KUKA KRL program: MyProgram_345().src

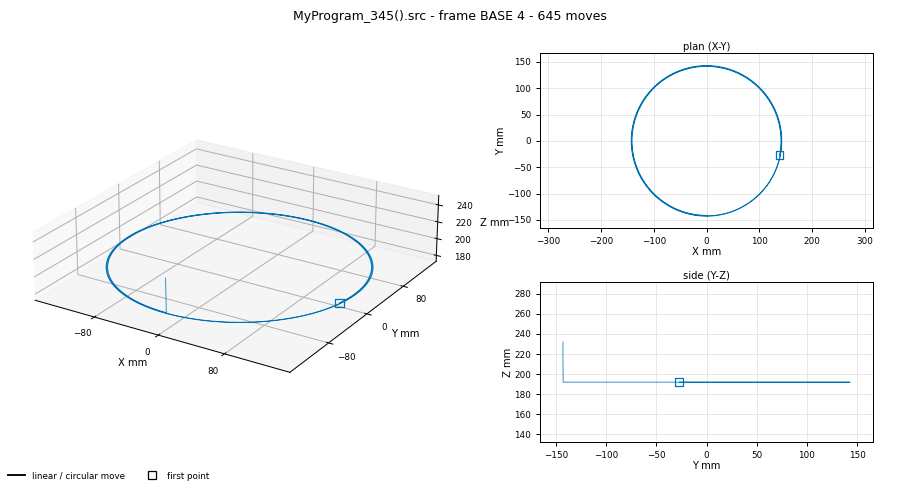
[picture p0: tool path of MyProgram_345().src in frame BASE 4, 645 of 645 moves have a stored position in this frame; points joined in program order, loops and branches not executed]
&ACCESS RVP
&REL 1
&PARAM TEMPLATE = C:\KRC\Roboter\Template\vorgabe
&PARAM EDITMASK = *
DEF MyProgram_345()
; ---- Setting reference (Base) ----
$BASE = BASE_DATA[4]

; --------------------------
; ---- Setting tool (TCP) ----
$TOOL = TOOL_DATA[3]
; --------------------------

$VEL.CP = VEL_APROX_PRINT
Startdeposition()
$VEL.CP = VEL_PRINT
LIN {X 138.5242,Y -27.3155,Z 192,A -4.5252,B 0.5611,C 0.0605,E1 0.722,E2 458.3283} C_DIS
LIN {X 139.2365,Y -23.4021,Z 192,A -3.481,B 0.5613,C 0.0586,E1 0.7225,E2 457.3622} C_DIS
LIN {X 139.7745,Y -19.9386,Z 192,A -2.1592,B 0.5617,C 0.0551,E1 0.7231,E2 456.0535} C_DIS
LIN {X 140.2586,Y -16.1943,Z 192,A -0.8679,B 0.562,C 0.052,E1 0.7235,E2 454.7945} C_DIS
LIN {X 140.6407,Y -12.4489,Z 192,A 0.376,B 0.5622,C 0.049,E1 0.7238,E2 453.5886} C_DIS
LIN {X 140.9254,Y -8.6325,Z 192,A 1.5623,B 0.5625,C 0.0463,E1 0.724,E2 452.4515} C_DIS
LIN {X 141.1118,Y -4.7394,Z 192,A 2.9278,B 0.5627,C 0.0429,E1 0.7241,E2 451.1146} C_DIS
LIN {X 141.1896,Y -0.6145,Z 192,A 4.1944,B 0.563,C 0.04,E1 0.7241,E2 449.9021} C_DIS
LIN {X 141.1462,Y 3.5236,Z 192,A 5.5812,B 0.5632,C 0.0366,E1 0.7241,E2 448.5537} C_DIS
LIN {X 140.9906,Y 7.504,Z 192,A 6.8322,B 0.5634,C 0.0338,E1 0.724,E2 447.3507} C_DIS
LIN {X 140.737,Y 11.3097,Z 192,A 8.1166,B 0.5635,C 0.0306,E1 0.7237,E2 446.1005} C_DIS
LIN {X 140.4091,Y 14.8267,Z 192,A 9.1787,B 0.5637,C 0.0283,E1 0.7234,E2 445.0867} C_DIS
LIN {X 140.0043,Y 18.2549,Z 192,A 10.3048,B 0.5637,C 0.0256,E1 0.7231,E2 443.996} C_DIS
LIN {X 139.3324,Y 22.8275,Z 192,A 12.3132,B 0.564,C 0.0198,E1 0.7222,E2 441.9693} C_DIS
LIN {X 138.4504,Y 27.6793,Z 192,A 14.134,B 0.5642,C 0.0151,E1 0.7212,E2 440.1713} C_DIS
LIN {X 137.041,Y 33.9819,Z 192,A 15.5668,B 0.5642,C 0.0131,E1 0.7204,E2 438.8911} C_DIS
LIN {X 135.2457,Y 40.5419,Z 192,A 17.9276,B 0.5643,C 0.0072,E1 0.7186,E2 436.5801} C_DIS
LIN {X 134.1293,Y 44.0907,Z 192,A 19.1032,B 0.5643,C 0.0045,E1 0.7176,E2 435.4462} C_DIS
LIN {X 132.9221,Y 47.6043,Z 192,A 20.2677,B 0.5643,C 0.0019,E1 0.7166,E2 434.3242} C_DIS
LIN {X 131.6486,Y 51.0197,Z 192,A 21.3577,B 0.5643,C -0.0004,E1 0.7155,E2 433.2822} C_DIS
LIN {X 130.3439,Y 54.2664,Z 192,A 22.5748,B 0.5643,C -0.0033,E1 0.7143,E2 432.0898} C_DIS
LIN {X 129.2468,Y 56.8363,Z 192,A 23.7777,B 0.5643,C -0.0067,E1 0.7129,E2 430.8782} C_DIS
LIN {X 127.791,Y 60.0377,Z 192,A 24.7987,B 0.5643,C -0.0087,E1 0.7118,E2 429.9068} C_DIS
LIN {X 126.0848,Y 63.5397,Z 192,A 26.0063,B 0.5643,C -0.0113,E1 0.7103,E2 428.7443} C_DIS
LIN {X 124.1773,Y 67.1944,Z 192,A 27.4129,B 0.5642,C -0.0146,E1 0.7085,E2 427.3696} C_DIS
LIN {X 122.0387,Y 71.0039,Z 192,A 28.7948,B 0.5641,C -0.0176,E1 0.7066,E2 426.0344} C_DIS
LIN {X 119.7699,Y 74.767,Z 192,A 30.2924,B 0.564,C -0.021,E1 0.7045,E2 424.5706} C_DIS
LIN {X 117.2837,Y 78.6098,Z 192,A 31.8113,B 0.5638,C -0.0243,E1 0.7022,E2 423.0915} C_DIS
LIN {X 114.6921,Y 82.3449,Z 192,A 33.3322,B 0.5637,C -0.0277,E1 0.6998,E2 421.6084} C_DIS
LIN {X 111.9551,Y 86.0294,Z 192,A 35.0251,B 0.5635,C -0.0316,E1 0.6969,E2 419.9352} C_DIS
LIN {X 109.8588,Y 88.6901,Z 192,A 35.9356,B 0.5634,C -0.0331,E1 0.6954,E2 419.0784} C_DIS
LIN {X 107.1281,Y 91.9702,Z 192,A 37.4224,B 0.5632,C -0.0364,E1 0.6927,E2 417.6197} C_DIS
LIN {X 104.0065,Y 95.4859,Z 192,A 38.9764,B 0.563,C -0.0395,E1 0.6899,E2 416.106} C_DIS
LIN {X 101.0756,Y 98.5838,Z 192,A 40.4488,B 0.5628,C -0.0426,E1 0.687,E2 414.6629} C_DIS
LIN {X 98.9534,Y 100.7132,Z 192,A 41.7136,B 0.5625,C -0.0455,E1 0.6845,E2 413.3929} C_DIS
LIN {X 95.9465,Y 103.5824,Z 192,A 42.79,B 0.5625,C -0.0471,E1 0.6824,E2 412.3852} C_DIS
LIN {X 93.0608,Y 106.1823,Z 192,A 44.1725,B 0.5622,C -0.05,E1 0.6795,E2 411.0242} C_DIS
LIN {X 89.4357,Y 109.2528,Z 192,A 45.7484,B 0.5619,C -0.0529,E1 0.6761,E2 409.4873} C_DIS
LIN {X 86.0148,Y 111.9663,Z 192,A 47.2728,B 0.5616,C -0.0558,E1 0.6728,E2 407.9901} C_DIS
LIN {X 82.3075,Y 114.7189,Z 192,A 48.8316,B 0.5613,C -0.0587,E1 0.6693,E2 406.4657} C_DIS
LIN {X 78.8287,Y 117.137,Z 192,A 50.2736,B 0.561,C -0.0612,E1 0.666,E2 405.0538} C_DIS
LIN {X 75.018,Y 119.6134,Z 192,A 51.8114,B 0.5607,C -0.0639,E1 0.6623,E2 403.549} C_DIS
LIN {X 71.2617,Y 121.8883,Z 192,A 53.3553,B 0.5604,C -0.0666,E1 0.6586,E2 402.0307} C_DIS
LIN {X 67.3753,Y 124.0788,Z 192,A 54.905,B 0.5601,C -0.0691,E1 0.6548,E2 400.5088} C_DIS
LIN {X 62.4464,Y 126.6285,Z 192,A 56.6735,B 0.5598,C -0.0718,E1 0.6504,E2 398.7912} C_DIS
LIN {X 59.695,Y 127.9495,Z 192,A 57.8562,B 0.5595,C -0.0738,E1 0.6474,E2 397.6145} C_DIS
LIN {X 56.3645,Y 129.4508,Z 192,A 59.1231,B 0.5593,C -0.0757,E1 0.6441,E2 396.3702} C_DIS
LIN {X 53.5399,Y 130.6464,Z 192,A 60.313,B 0.559,C -0.0776,E1 0.641,E2 395.1862} C_DIS
LIN {X 49.9685,Y 132.052,Z 192,A 61.5782,B 0.5588,C -0.0793,E1 0.6377,E2 393.9512} C_DIS
LIN {X 46.7273,Y 133.2336,Z 192,A 62.8545,B 0.5585,C -0.0811,E1 0.6342,E2 392.6878} C_DIS
LIN {X 43.1768,Y 134.4254,Z 192,A 64.2206,B 0.5582,C -0.083,E1 0.6306,E2 391.3377} C_DIS
LIN {X 35.1127,Y 136.754,Z 192,A 67.1312,B 0.5577,C -0.0866,E1 0.6226,E2 388.478} C_DIS
LIN {X 28.547,Y 138.2738,Z 192,A 69.6083,B 0.5572,C -0.0895,E1 0.6157,E2 386.0273} C_DIS
LIN {X 23.8823,Y 139.1564,Z 192,A 71.397,B 0.5569,C -0.0915,E1 0.6107,E2 384.2529} C_DIS
LIN {X 20.3949,Y 139.7092,Z 192,A 72.6632,B 0.5567,C -0.0928,E1 0.6071,E2 383.0035} C_DIS
LIN {X 17.2318,Y 140.1349,Z 192,A 73.8305,B 0.5565,C -0.0939,E1 0.6038,E2 381.8492} C_DIS
LIN {X 13.6174,Y 140.5313,Z 192,A 75.1425,B 0.5563,C -0.0951,E1 0.6001,E2 380.5536} C_DIS
LIN {X 9.6219,Y 140.8628,Z 192,A 76.7148,B 0.5561,C -0.0966,E1 0.5955,E2 378.9872} C_DIS
LIN {X 5.5113,Y 141.0819,Z 192,A 78.1803,B 0.5559,C -0.0977,E1 0.5913,E2 377.5421} C_DIS
LIN {X 1.1101,Y 141.1856,Z 192,A 79.8215,B 0.5556,C -0.0988,E1 0.5866,E2 375.9156} C_DIS
LIN {X -2.5499,Y 141.1667,Z 192,A 81.2212,B 0.5555,C -0.0998,E1 0.5826,E2 374.5247} C_DIS
LIN {X -6.4253,Y 141.0448,Z 192,A 82.7609,B 0.5553,C -0.1008,E1 0.5781,E2 372.9889} C_DIS
LIN {X -10.1902,Y 140.8213,Z 192,A 84.1527,B 0.5552,C -0.1015,E1 0.5741,E2 371.6108} C_DIS
LIN {X -13.9892,Y 140.4956,Z 192,A 85.4332,B 0.5551,C -0.102,E1 0.5705,E2 370.3563} C_DIS
LIN {X -18.5339,Y 139.9678,Z 192,A 87.497,B 0.5549,C -0.1031,E1 0.5645,E2 368.2736} C_DIS
LIN {X -22.8627,Y 139.3265,Z 192,A 89.1306,B 0.5548,C -0.1036,E1 0.5598,E2 366.6543} C_DIS
LIN {X -26.405,Y 138.6983,Z 192,A 90.5233,B 0.5548,C -0.1039,E1 0.5559,E2 365.2685} C_DIS
LIN {X -29.884,Y 137.9904,Z 192,A 91.948,B 0.5547,C -0.1042,E1 0.5518,E2 363.846} C_DIS
LIN {X -33.9548,Y 137.0478,Z 192,A 93.7775,B 0.5546,C -0.1046,E1 0.5466,E2 362.0046} C_DIS
LIN {X -38.0062,Y 135.9776,Z 192,A 95.319,B 0.5546,C -0.1046,E1 0.5423,E2 360.4788} C_DIS
LIN {X -41.3069,Y 135.0115,Z 192,A 96.5979,B 0.5546,C -0.1044,E1 0.5388,E2 359.2116} C_DIS
LIN {X -44.3383,Y 134.0469,Z 192,A 97.9917,B 0.5546,C -0.1044,E1 0.5349,E2 357.8086} C_DIS
LIN {X -47.0982,Y 133.1045,Z 192,A 99.3629,B 0.5546,C -0.1044,E1 0.5311,E2 356.4203} C_DIS
LIN {X -50.6134,Y 131.8066,Z 192,A 100.8481,B 0.5547,C -0.104,E1 0.527,E2 354.9391} C_DIS
LIN {X -53.6288,Y 130.6102,Z 192,A 102.5352,B 0.5547,C -0.1038,E1 0.5224,E2 353.2173} C_DIS
LIN {X -57.197,Y 129.0856,Z 192,A 103.7496,B 0.5549,C -0.1031,E1 0.5193,E2 352.038} C_DIS
LIN {X -60.1404,Y 127.7424,Z 192,A 105.2375,B 0.5549,C -0.1026,E1 0.5153,E2 350.5342} C_DIS
LIN {X -64.6568,Y 125.516,Z 192,A 107.3683,B 0.5552,C -0.1015,E1 0.5097,E2 348.396} C_DIS
LIN {X -67.4098,Y 124.06,Z 192,A 109.262,B 0.5552,C -0.1009,E1 0.5048,E2 346.4422} C_DIS
LIN {X -71.8848,Y 121.5223,Z 192,A 110.9515,B 0.5556,C -0.0993,E1 0.5006,E2 344.7923} C_DIS
LIN {X -75.7994,Y 119.1197,Z 192,A 112.9667,B 0.5558,C -0.0978,E1 0.4956,E2 342.7635} C_DIS
LIN {X -79.6799,Y 116.5594,Z 192,A 115.3227,B 0.5561,C -0.0961,E1 0.4899,E2 340.3627} C_DIS
LIN {X -82.7739,Y 114.3826,Z 192,A 116.7096,B 0.5564,C -0.0946,E1 0.4866,E2 338.9912} C_DIS
LIN {X -86.4509,Y 111.6295,Z 192,A 118.7765,B 0.5567,C -0.0925,E1 0.4818,E2 336.9053} C_DIS
LIN {X -90.153,Y 108.6616,Z 192,A 120.8713,B 0.5571,C -0.0902,E1 0.4771,E2 334.7948} C_DIS
LIN {X -93.2484,Y 106.0177,Z 192,A 122.8335,B 0.5575,C -0.088,E1 0.4728,E2 332.8028} C_DIS
LIN {X -96.6151,Y 102.959,Z 192,A 124.9266,B 0.5579,C -0.0854,E1 0.4683,E2 330.686} C_DIS
LIN {X -99.7496,Y 99.9251,Z 192,A 126.9433,B 0.5583,C -0.0827,E1 0.4641,E2 328.6454} C_DIS
LIN {X -102.8714,Y 96.708,Z 192,A 129.0955,B 0.5587,C -0.0797,E1 0.4598,E2 326.4604} C_DIS
LIN {X -105.9836,Y 93.287,Z 192,A 131.2873,B 0.5592,C -0.0764,E1 0.4555,E2 324.2373} C_DIS
LIN {X -108.8114,Y 89.9722,Z 192,A 133.4193,B 0.5596,C -0.073,E1 0.4515,E2 322.0688} C_DIS
LIN {X -111.9551,Y 86.0294,Z 192,A 136.4707,B 0.5602,C -0.0683,E1 0.446,E2 318.9128} C_DIS
LIN {X -114.7818,Y 82.2196,Z 192,A 138.1377,B 0.5606,C -0.065,E1 0.4432,E2 317.2743} C_DIS
LIN {X -117.5668,Y 78.1857,Z 192,A 140.6425,B 0.5611,C -0.0605,E1 0.4391,E2 314.7156} C_DIS
LIN {X -119.9857,Y 74.4203,Z 192,A 142.6975,B 0.5615,C -0.0565,E1 0.4359,E2 312.636} C_DIS
LIN {X -123.2884,Y 68.8117,Z 192,A 146.2773,B 0.5622,C -0.0496,E1 0.4307,E2 308.9552} C_DIS
LIN {X -125.6023,Y 64.4874,Z 192,A 148.651,B 0.5626,C -0.0446,E1 0.4275,E2 306.5401} C_DIS
LIN {X -127.9588,Y 59.6746,Z 192,A 151.6555,B 0.5631,C -0.0383,E1 0.4237,E2 303.4432} C_DIS
LIN {X -129.8067,Y 55.5407,Z 192,A 154.0352,B 0.5634,C -0.0331,E1 0.421,E2 301.0026} C_DIS
LIN {X -131.5415,Y 51.2953,Z 192,A 155.8705,B 0.5636,C -0.0286,E1 0.419,E2 299.1713} C_DIS
LIN {X -132.5169,Y 48.7273,Z 192,A 157.7152,B 0.5638,C -0.0246,E1 0.4171,E2 297.2425} C_DIS
LIN {X -133.9593,Y 44.6014,Z 192,A 159.9336,B 0.564,C -0.0194,E1 0.4151,E2 294.9728} C_DIS
LIN {X -134.9324,Y 41.5656,Z 192,A 161.7041,B 0.5642,C -0.0153,E1 0.4135,E2 293.1463} C_DIS
LIN {X -135.8406,Y 38.4962,Z 192,A 163.2032,B 0.5642,C -0.0115,E1 0.4123,E2 291.6241} C_DIS
LIN {X -136.6138,Y 35.6597,Z 192,A 165.5888,B 0.5643,C -0.0063,E1 0.4106,E2 289.0943} C_DIS
LIN {X -137.591,Y 31.6731,Z 192,A 166.8745,B 0.5643,C -0.0025,E1 0.4097,E2 287.8561} C_DIS
LIN {X -138.5269,Y 27.3017,Z 192,A 169.7946,B 0.5643,C 0.0043,E1 0.408,E2 284.8005} C_DIS
LIN {X -139.6213,Y 20.9931,Z 192,A 173.1218,B 0.5643,C 0.0128,E1 0.4064,E2 281.3831} C_DIS
LIN {X -140.228,Y 16.451,Z 192,A 175.5869,B 0.5641,C 0.019,E1 0.4055,E2 278.8419} C_DIS
LIN {X -140.6546,Y 12.2842,Z 192,A 178.0252,B 0.5638,C 0.0251,E1 0.4049,E2 276.3092} C_DIS
LIN {X -140.8877,Y 9.2448,Z 192,A -179.8372,B 0.5636,C 0.0302,E1 0.4045,E2 274.0544} C_DIS
LIN {X -141.0977,Y 5.1076,Z 192,A -178.0006,B 0.5633,C 0.0352,E1 0.4043,E2 272.1982} C_DIS
LIN {X -141.1833,Y -1.537,Z 192,A -174.4443,B 0.5626,C 0.0443,E1 0.4043,E2 268.5288} C_DIS
LIN {X -141.0589,Y -6.1025,Z 192,A -171.3976,B 0.562,C 0.0516,E1 0.4046,E2 265.321} C_DIS
LIN {X -140.8113,Y -10.3266,Z 192,A -168.6963,B 0.5614,C 0.0581,E1 0.4052,E2 262.4846} C_DIS
LIN {X -140.2534,Y -16.2384,Z 192,A -166.4993,B 0.5607,C 0.0644,E1 0.4058,E2 260.3184} C_DIS
LIN {X -139.8061,Y -19.7168,Z 192,A -164.5222,B 0.5601,C 0.0692,E1 0.4066,E2 258.2647} C_DIS
LIN {X -138.8649,Y -25.5228,Z 192,A -161.2506,B 0.5591,C 0.0772,E1 0.4082,E2 254.8696} C_DIS
LIN {X -138.0677,Y -29.5261,Z 192,A -159.1217,B 0.5583,C 0.0824,E1 0.4095,E2 252.6741} C_DIS
LIN {X -137.2735,Y -33.0212,Z 192,A -157.251,B 0.5576,C 0.0869,E1 0.4107,E2 250.7444} C_DIS
LIN {X -136.3362,Y -36.7007,Z 192,A -155.2273,B 0.5569,C 0.0916,E1 0.4122,E2 248.6517} C_DIS
LIN {X -135.1685,Y -40.794,Z 192,A -152.8988,B 0.556,C 0.097,E1 0.4141,E2 246.2365} C_DIS
LIN {X -134.1293,Y -44.0907,Z 192,A -150.6088,B 0.5551,C 0.1018,E1 0.4162,E2 243.8168} C_DIS
LIN {X -132.8674,Y -47.7561,Z 192,A -149.3984,B 0.5545,C 0.1052,E1 0.4173,E2 242.6605} C_DIS
LIN {X -131.7622,Y -50.7275,Z 192,A -147.3606,B 0.5537,C 0.1093,E1 0.4194,E2 240.5122} C_DIS
LIN {X -130.6124,Y -53.6235,Z 192,A -145.81,B 0.553,C 0.1127,E1 0.4211,E2 238.9196} C_DIS
LIN {X -128.8353,Y -57.7566,Z 192,A -143.4773,B 0.552,C 0.1176,E1 0.4238,E2 236.5116} C_DIS
LIN {X -127.4653,Y -60.7203,Z 192,A -141.7834,B 0.5512,C 0.1211,E1 0.4259,E2 234.7627} C_DIS
LIN {X -125.8921,Y -63.9181,Z 192,A -140.0703,B 0.5504,C 0.1246,E1 0.4282,E2 233.0098} C_DIS
LIN {X -124.1723,Y -67.2036,Z 192,A -137.9104,B 0.5495,C 0.1286,E1 0.4312,E2 230.7509} C_DIS
LIN {X -121.9679,Y -71.1262,Z 192,A -135.6323,B 0.5485,C 0.1329,E1 0.4345,E2 228.4043} C_DIS
LIN {X -119.5569,Y -75.1076,Z 192,A -133.347,B 0.5475,C 0.1371,E1 0.438,E2 226.0584} C_DIS
LIN {X -117.1181,Y -78.8567,Z 192,A -131.1217,B 0.5465,C 0.1409,E1 0.4416,E2 223.7703} C_DIS
LIN {X -114.5576,Y -82.5325,Z 192,A -129.0173,B 0.5456,C 0.1445,E1 0.4451,E2 221.6218} C_DIS
LIN {X -109.5938,Y -89.0184,Z 192,A -124.9502,B 0.5439,C 0.1508,E1 0.4525,E2 217.4383} C_DIS
LIN {X -105.9183,Y -93.3609,Z 192,A -122.2264,B 0.5428,C 0.1547,E1 0.4577,E2 214.6496} C_DIS
LIN {X -102.9112,Y -96.6658,Z 192,A -120.1081,B 0.5419,C 0.1575,E1 0.4619,E2 212.4835} C_DIS
LIN {X -96.5479,Y -103.0223,Z 192,A -115.9063,B 0.5404,C 0.1627,E1 0.4707,E2 208.1948} C_DIS
LIN {X -93.1478,Y -106.1064,Z 192,A -113.9445,B 0.5397,C 0.165,E1 0.475,E2 206.2172} C_DIS
LIN {X -89.5276,Y -109.1777,Z 192,A -111.6621,B 0.539,C 0.1672,E1 0.4802,E2 203.8783} C_DIS
LIN {X -86.0232,Y -111.9598,Z 192,A -109.6421,B 0.5384,C 0.1691,E1 0.4849,E2 201.8256} C_DIS
LIN {X -82.3935,Y -114.6574,Z 192,A -107.5945,B 0.5379,C 0.1709,E1 0.4897,E2 199.7438} C_DIS
LIN {X -78.7099,Y -117.2169,Z 192,A -105.619,B 0.5374,C 0.1724,E1 0.4945,E2 197.7432} C_DIS
LIN {X -75.0257,Y -119.6086,Z 192,A -103.6912,B 0.537,C 0.1737,E1 0.4993,E2 195.7919} C_DIS
LIN {X -71.1828,Y -121.9346,Z 192,A -101.7704,B 0.5366,C 0.1749,E1 0.5041,E2 193.8549} C_DIS
LIN {X -67.3853,Y -124.0734,Z 192,A -99.7334,B 0.5363,C 0.1758,E1 0.5094,E2 191.7744} C_DIS
LIN {X -62.7554,Y -126.4761,Z 192,A -97.6185,B 0.5359,C 0.1769,E1 0.5149,E2 189.6592} C_DIS
LIN {X -58.5907,Y -128.4601,Z 192,A -95.6908,B 0.5357,C 0.1776,E1 0.52,E2 187.7221} C_DIS
LIN {X -54.4999,Y -130.2463,Z 192,A -93.9571,B 0.5355,C 0.1783,E1 0.5246,E2 186.0001} C_DIS
LIN {X -51.2884,Y -131.5442,Z 192,A -92.4968,B 0.5354,C 0.1786,E1 0.5286,E2 184.5306} C_DIS
LIN {X -47.9773,Y -132.7876,Z 192,A -91.0696,B 0.5353,C 0.1788,E1 0.5325,E2 183.1041} C_DIS
LIN {X -43.9542,Y -134.1748,Z 192,A -88.7402,B 0.5355,C 0.1782,E1 0.5392,E2 180.6769} C_DIS
LIN {X -39.3274,Y -135.6019,Z 192,A -87.2994,B 0.5353,C 0.1789,E1 0.543,E2 179.3199} C_DIS
LIN {X -35.2083,Y -136.7297,Z 192,A -85.1679,B 0.5355,C 0.1781,E1 0.5492,E2 177.1233} C_DIS
LIN {X -31.0454,Y -137.7344,Z 192,A -83.8745,B 0.5354,C 0.1786,E1 0.5527,E2 175.9008} C_DIS
LIN {X -26.8167,Y -138.6196,Z 192,A -82.1983,B 0.5354,C 0.1783,E1 0.5574,E2 174.2361} C_DIS
LIN {X -23.2817,Y -139.2566,Z 192,A -80.7844,B 0.5356,C 0.1779,E1 0.5614,E2 172.8285} C_DIS
LIN {X -19.8588,Y -139.7858,Z 192,A -79.3969,B 0.5358,C 0.1774,E1 0.5654,E2 171.4432} C_DIS
LIN {X -15.7219,Y -140.3127,Z 192,A -77.8099,B 0.5359,C 0.1769,E1 0.57,E2 169.8722} C_DIS
LIN {X -12.0026,Y -140.6784,Z 192,A -76.3454,B 0.5362,C 0.1762,E1 0.5742,E2 168.4152} C_DIS
LIN {X -8.8272,Y -140.9134,Z 192,A -75.0655,B 0.5364,C 0.1754,E1 0.5779,E2 167.1365} C_DIS
LIN {X -4.3497,Y -141.1232,Z 192,A -73.3263,B 0.5367,C 0.1744,E1 0.5829,E2 165.409} C_DIS
LIN {X -0.1029,Y -141.1912,Z 192,A -71.7287,B 0.5371,C 0.1734,E1 0.5875,E2 163.8306} C_DIS
LIN {X -0.1029,Y -141.1912,Z 192,A -71.7287,B 0.5371,C 0.1734,E1 0.5875,E2 163.8306} C_DIS
Enddeposition()
LIN {X 1.0199,Y -142.0827,Z 192,A -71.4245,B 0.537,C 0.1736,E1 0.5882,E2 163.5677} C_DIS
Startdeposition()
$VEL.CP = VEL_PRINT
LIN {X -3.1233,Y -142.0562,Z 192,A -73.5823,B 0.5362,C 0.176,E1 0.5817,E2 165.8051} C_DIS
LIN {X -6.8466,Y -141.9237,Z 192,A -74.8566,B 0.5361,C 0.1765,E1 0.5781,E2 167.0436} C_DIS
LIN {X -9.8472,Y -141.7477,Z 192,A -76.1523,B 0.5358,C 0.1774,E1 0.5743,E2 168.3535} C_DIS
LIN {X -14.4877,Y -141.3496,Z 192,A -77.7778,B 0.5356,C 0.1778,E1 0.5697,E2 169.9394} C_DIS
LIN {X -18.6545,Y -140.8586,Z 192,A -79.5013,B 0.5353,C 0.1787,E1 0.5648,E2 171.669} C_DIS
LIN {X -22.3643,Y -140.3186,Z 192,A -80.8938,B 0.5353,C 0.179,E1 0.5608,E2 173.043} C_DIS
LIN {X -24.9898,Y -139.8734,Z 192,A -82.0034,B 0.5351,C 0.1794,E1 0.5576,E2 174.159} C_DIS
LIN {X -29.2238,Y -139.0526,Z 192,A -83.6255,B 0.5351,C 0.1796,E1 0.553,E2 175.7631} C_DIS
LIN {X -32.0395,Y -138.4294,Z 192,A -84.8401,B 0.5349,C 0.1799,E1 0.5496,E2 176.9866} C_DIS
LIN {X -35.089,Y -137.6874,Z 192,A -86.0904,B 0.5349,C 0.18,E1 0.546,E2 178.235} C_DIS
LIN {X -38.3299,Y -136.8205,Z 192,A -87.4611,B 0.5349,C 0.1801,E1 0.5422,E2 179.6092} C_DIS
LIN {X -42.821,Y -135.4827,Z 192,A -89.141,B 0.5349,C 0.1798,E1 0.5376,E2 181.256} C_DIS
LIN {X -47.2474,Y -134.0047,Z 192,A -91.171,B 0.5349,C 0.1798,E1 0.5319,E2 183.3107} C_DIS
LIN {X -49.9377,Y -133.0234,Z 192,A -92.4033,B 0.5349,C 0.1797,E1 0.5285,E2 184.556} C_DIS
LIN {X -53.1954,Y -131.7545,Z 192,A -93.8591,B 0.5351,C 0.1794,E1 0.5246,E2 186.0197} C_DIS
LIN {X -57.3886,Y -129.9846,Z 192,A -95.6365,B 0.5353,C 0.1787,E1 0.5198,E2 187.7884} C_DIS
LIN {X -60.2323,Y -128.6914,Z 192,A -97.0055,B 0.5354,C 0.1783,E1 0.5162,E2 189.1754} C_DIS
LIN {X -63.1297,Y -127.2938,Z 192,A -98.3855,B 0.5356,C 0.1778,E1 0.5125,E2 190.5691} C_DIS
LIN {X -66.448,Y -125.5939,Z 192,A -99.9507,B 0.5359,C 0.177,E1 0.5085,E2 192.1447} C_DIS
LIN {X -70.1242,Y -123.5809,Z 192,A -101.88,B 0.5362,C 0.1762,E1 0.5035,E2 194.1129} C_DIS
LIN {X -74.1762,Y -121.1918,Z 192,A -103.8721,B 0.5366,C 0.1749,E1 0.4985,E2 196.1206} C_DIS
LIN {X -77.9071,Y -118.8281,Z 192,A -105.821,B 0.537,C 0.1735,E1 0.4937,E2 198.0967} C_DIS
LIN {X -81.7579,Y -116.212,Z 192,A -107.8571,B 0.5375,C 0.1719,E1 0.4887,E2 200.1585} C_DIS
LIN {X -85.4635,Y -113.5146,Z 192,A -109.8463,B 0.5381,C 0.1701,E1 0.4841,E2 202.1704} C_DIS
LIN {X -88.9199,Y -110.8284,Z 192,A -111.8567,B 0.5387,C 0.1682,E1 0.4794,E2 204.2201} C_DIS
LIN {X -92.0421,Y -108.2487,Z 192,A -113.5883,B 0.5393,C 0.1663,E1 0.4755,E2 205.9674} C_DIS
LIN {X -95.1246,Y -105.5512,Z 192,A -115.5912,B 0.5399,C 0.1643,E1 0.4711,E2 208.0262} C_DIS
LIN {X -98.181,Y -102.7133,Z 192,A -117.405,B 0.5406,C 0.162,E1 0.4672,E2 209.8608} C_DIS
LIN {X -101.7504,Y -99.1796,Z 192,A -119.839,B 0.5415,C 0.1591,E1 0.4622,E2 212.3593} C_DIS
LIN {X -104.9251,Y -95.8148,Z 192,A -122.0269,B 0.5423,C 0.1562,E1 0.4578,E2 214.5978} C_DIS
LIN {X -108.106,Y -92.21,Z 192,A -123.9147,B 0.5432,C 0.1531,E1 0.4542,E2 216.4775} C_DIS
LIN {X -109.8966,Y -90.0685,Z 192,A -125.5791,B 0.5438,C 0.1509,E1 0.451,E2 218.2261} C_DIS
LIN {X -112.6158,Y -86.6453,Z 192,A -127.8845,B 0.5447,C 0.1476,E1 0.4468,E2 220.6157} C_DIS
LIN {X -115.8068,Y -82.3315,Z 192,A -130.3452,B 0.5458,C 0.1434,E1 0.4426,E2 223.1221} C_DIS
LIN {X -118.4142,Y -78.5354,Z 192,A -132.5927,B 0.5469,C 0.1395,E1 0.439,E2 225.4295} C_DIS
LIN {X -120.7608,Y -74.8761,Z 192,A -134.7185,B 0.5478,C 0.1357,E1 0.4356,E2 227.6121} C_DIS
LIN {X -122.9723,Y -71.1854,Z 192,A -136.8636,B 0.5488,C 0.1317,E1 0.4324,E2 229.8195} C_DIS
LIN {X -125.0902,Y -67.3946,Z 192,A -139.0654,B 0.5498,C 0.1275,E1 0.4293,E2 232.0895} C_DIS
LIN {X -126.8397,Y -64.0382,Z 192,A -140.9713,B 0.5506,C 0.1237,E1 0.4268,E2 234.0523} C_DIS
LIN {X -129.0616,Y -59.4318,Z 192,A -144.1165,B 0.552,C 0.1177,E1 0.4229,E2 237.3592} C_DIS
LIN {X -130.8601,Y -55.3629,Z 192,A -145.7078,B 0.5528,C 0.1137,E1 0.4211,E2 238.9197} C_DIS
LIN {X -131.9054,Y -52.8211,Z 192,A -147.1641,B 0.5534,C 0.1106,E1 0.4195,E2 240.4275} C_DIS
LIN {X -132.8818,Y -50.316,Z 192,A -148.5042,B 0.554,C 0.1076,E1 0.4181,E2 241.8052} C_DIS
LIN {X -133.8675,Y -47.6323,Z 192,A -150.1002,B 0.5547,C 0.1042,E1 0.4165,E2 243.4661} C_DIS
LIN {X -134.9501,Y -44.4711,Z 192,A -151.909,B 0.5554,C 0.1002,E1 0.4148,E2 245.3421} C_DIS
LIN {X -135.9994,Y -41.151,Z 192,A -153.6933,B 0.5561,C 0.096,E1 0.4133,E2 247.1812} C_DIS
LIN {X -136.8752,Y -38.1344,Z 192,A -155.3604,B 0.5568,C 0.0922,E1 0.412,E2 248.906} C_DIS
LIN {X -137.9184,Y -34.1788,Z 192,A -157.5471,B 0.5576,C 0.087,E1 0.4104,E2 251.1693} C_DIS
LIN {X -138.7239,Y -30.7462,Z 192,A -159.4054,B 0.5583,C 0.0826,E1 0.4092,E2 253.0894} C_DIS
LIN {X -139.5958,Y -26.4975,Z 192,A -161.7055,B 0.5591,C 0.077,E1 0.4079,E2 255.467} C_DIS
LIN {X -140.1758,Y -23.2343,Z 192,A -163.6258,B 0.5597,C 0.0724,E1 0.4069,E2 257.4688} C_DIS
LIN {X -140.8224,Y -18.9307,Z 192,A -166.0269,B 0.5604,C 0.0665,E1 0.406,E2 259.9592} C_DIS
LIN {X -141.3316,Y -14.655,Z 192,A -168.4104,B 0.5611,C 0.0605,E1 0.4052,E2 262.4311} C_DIS
LIN {X -141.7694,Y -9.5469,Z 192,A -171.1724,B 0.5618,C 0.0536,E1 0.4046,E2 265.2868} C_DIS
LIN {X -141.9542,Y -6.2126,Z 192,A -172.7429,B 0.5622,C 0.0494,E1 0.4044,E2 266.8869} C_DIS
LIN {X -142.0572,Y -3.0617,Z 192,A -174.6195,B 0.5626,C 0.0448,E1 0.4042,E2 268.8442} C_DIS
LIN {X -142.0915,Y 0.1202,Z 192,A -176.5729,B 0.5629,C 0.04,E1 0.4042,E2 270.886} C_DIS
LIN {X -142.0103,Y 4.7738,Z 192,A -178.7666,B 0.5633,C 0.0341,E1 0.4043,E2 273.1204} C_DIS
LIN {X -141.857,Y 8.1297,Z 192,A 179.4826,B 0.5636,C 0.0296,E1 0.4046,E2 274.9223} C_DIS
LIN {X -141.5949,Y 11.8332,Z 192,A 177.4706,B 0.5638,C 0.0245,E1 0.405,E2 277.0001} C_DIS
LIN {X -141.3578,Y 14.4119,Z 192,A 175.9655,B 0.564,C 0.0208,E1 0.4055,E2 278.564} C_DIS
LIN {X -141.069,Y 16.9903,Z 192,A 174.5098,B 0.5641,C 0.0171,E1 0.4059,E2 280.0712} C_DIS
LIN {X -140.5426,Y 20.9154,Z 192,A 171.6614,B 0.5643,C 0.0104,E1 0.4072,E2 283.0758} C_DIS
LIN {X -139.8038,Y 25.3789,Z 192,A 169.801,B 0.5643,C 0.0054,E1 0.4081,E2 284.9395} C_DIS
LIN {X -138.5248,Y 31.6216,Z 192,A 166.8365,B 0.5643,C -0.0022,E1 0.4098,E2 287.9511} C_DIS
LIN {X -136.9663,Y 37.8086,Z 192,A 163.284,B 0.5643,C -0.0108,E1 0.4123,E2 291.6213} C_DIS
LIN {X -136.9663,Y 37.8086,Z 192,A 163.2828,B 0.5643,C -0.0108,E1 0.4123,E2 291.6227} C_DIS
LIN {X -136.099,Y 40.8253,Z 192,A 161.4573,B 0.5642,C -0.015,E1 0.4138,E2 293.5144} C_DIS
LIN {X -135.2129,Y 43.6655,Z 192,A 159.7139,B 0.564,C -0.019,E1 0.4154,E2 295.3211} C_DIS
LIN {X -134.0258,Y 47.1864,Z 192,A 157.9049,B 0.5639,C -0.0233,E1 0.4171,E2 297.1656} C_DIS
LIN {X -132.7111,Y 50.7676,Z 192,A 155.926,B 0.5637,C -0.0279,E1 0.4191,E2 299.1947} C_DIS
LIN {X -131.6564,Y 53.4387,Z 192,A 154.447,B 0.5635,C -0.0312,E1 0.4206,E2 300.7098} C_DIS
LIN {X -130.1901,Y 56.9198,Z 192,A 152.3791,B 0.5632,C -0.0357,E1 0.423,E2 302.8386} C_DIS
LIN {X -127.3087,Y 63.0995,Z 192,A 148.8679,B 0.5627,C -0.0432,E1 0.4274,E2 306.4334} C_DIS
LIN {X -127.3087,Y 63.0995,Z 192,A 148.867,B 0.5627,C -0.0432,E1 0.4274,E2 306.4345} C_DIS
LIN {X -125.4548,Y 66.7129,Z 192,A 146.8543,B 0.5624,C -0.0475,E1 0.43,E2 308.4877} C_DIS
LIN {X -123.2816,Y 70.649,Z 192,A 144.77,B 0.562,C -0.0518,E1 0.433,E2 310.6006} C_DIS
LIN {X -120.6271,Y 75.091,Z 192,A 141.8532,B 0.5615,C -0.0572,E1 0.4374,E2 313.6058} C_DIS
LIN {X -118.2496,Y 78.7821,Z 192,A 139.6255,B 0.561,C -0.0613,E1 0.4409,E2 315.881} C_DIS
LIN {X -115.8508,Y 82.27,Z 192,A 137.4459,B 0.5606,C -0.0652,E1 0.4446,E2 318.1091} C_DIS
LIN {X -112.8748,Y 86.3066,Z 192,A 135.4202,B 0.5601,C -0.0689,E1 0.448,E2 320.134} C_DIS
LIN {X -111.0516,Y 88.6405,Z 192,A 133.6917,B 0.5598,C -0.0716,E1 0.4512,E2 321.917} C_DIS
LIN {X -108.3045,Y 91.9766,Z 192,A 131.6001,B 0.5594,C -0.0749,E1 0.4551,E2 324.0433} C_DIS
LIN {X -105.3777,Y 95.316,Z 192,A 129.4346,B 0.5589,C -0.0781,E1 0.4593,E2 326.2457} C_DIS
LIN {X -102.211,Y 98.7041,Z 192,A 127.2773,B 0.5585,C -0.0812,E1 0.4636,E2 328.4307} C_DIS
LIN {X -99.0546,Y 101.8716,Z 192,A 125.1787,B 0.5581,C -0.084,E1 0.468,E2 330.5577} C_DIS
LIN {X -95.7633,Y 104.9718,Z 192,A 123.1444,B 0.5577,C -0.0866,E1 0.4723,E2 332.6118} C_DIS
LIN {X -92.4531,Y 107.8985,Z 192,A 121.0661,B 0.5573,C -0.089,E1 0.4769,E2 334.7181} C_DIS
LIN {X -89.0781,Y 110.7008,Z 192,A 119.091,B 0.557,C -0.0912,E1 0.4814,E2 336.7123} C_DIS
LIN {X -85.4109,Y 113.5543,Z 192,A 116.9748,B 0.5566,C -0.0932,E1 0.4863,E2 338.8509} C_DIS
LIN {X -81.5461,Y 116.3611,Z 192,A 114.9198,B 0.5563,C -0.0952,E1 0.4912,E2 340.9172} C_DIS
LIN {X -78.3242,Y 118.5535,Z 192,A 113.2013,B 0.556,C -0.0966,E1 0.4953,E2 342.649} C_DIS
LIN {X -75.0305,Y 120.6647,Z 192,A 111.4877,B 0.5558,C -0.0979,E1 0.4996,E2 344.3747} C_DIS
LIN {X -71.531,Y 122.7723,Z 192,A 109.6726,B 0.5556,C -0.099,E1 0.5042,E2 346.2049} C_DIS
LIN {X -67.1356,Y 125.2293,Z 192,A 107.5839,B 0.5554,C -0.1003,E1 0.5095,E2 348.2981} C_DIS
LIN {X -63.8334,Y 126.9439,Z 192,A 105.7297,B 0.5552,C -0.101,E1 0.5144,E2 350.1846} C_DIS
LIN {X -58.8005,Y 129.3531,Z 192,A 103.6365,B 0.5551,C -0.1021,E1 0.5198,E2 352.2621} C_DIS
LIN {X -55.9517,Y 130.6086,Z 192,A 102.3545,B 0.555,C -0.1025,E1 0.5233,E2 353.5459} C_DIS
LIN {X -52.7649,Y 131.928,Z 192,A 100.9748,B 0.5549,C -0.1029,E1 0.527,E2 354.924} C_DIS
LIN {X -49.372,Y 133.2353,Z 192,A 99.3859,B 0.5549,C -0.1032,E1 0.5313,E2 356.5236} C_DIS
LIN {X -45.7954,Y 134.5081,Z 192,A 97.8984,B 0.5549,C -0.1034,E1 0.5354,E2 358.0065} C_DIS
LIN {X -42.9152,Y 135.4527,Z 192,A 96.6692,B 0.5548,C -0.1034,E1 0.5388,E2 359.2357} C_DIS
LIN {X -39.735,Y 136.4192,Z 192,A 95.3255,B 0.5548,C -0.1035,E1 0.5426,E2 360.5791} C_DIS
LIN {X -35.879,Y 137.4857,Z 192,A 93.7137,B 0.5548,C -0.1034,E1 0.5471,E2 362.1901} C_DIS
LIN {X -31.4991,Y 138.5528,Z 192,A 91.7702,B 0.5548,C -0.103,E1 0.5526,E2 364.1445} C_DIS
LIN {X -27.7547,Y 139.3524,Z 192,A 90.4363,B 0.5549,C -0.1029,E1 0.5564,E2 365.4582} C_DIS
LIN {X -25.0006,Y 139.8715,Z 192,A 89.4032,B 0.5549,C -0.1027,E1 0.5593,E2 366.4817} C_DIS
LIN {X -22.3749,Y 140.317,Z 192,A 88.3558,B 0.555,C -0.1023,E1 0.5623,E2 367.5262} C_DIS
LIN {X -19.2353,Y 140.7825,Z 192,A 86.9346,B 0.5551,C -0.1016,E1 0.5665,E2 368.9603} C_DIS
LIN {X -15.2091,Y 141.272,Z 192,A 85.6203,B 0.5551,C -0.1013,E1 0.5702,E2 370.2435} C_DIS
LIN {X -12.3042,Y 141.5551,Z 192,A 84.3967,B 0.5553,C -0.1006,E1 0.5737,E2 371.4711} C_DIS
LIN {X -9.3063,Y 141.7845,Z 192,A 83.2569,B 0.5554,C -0.1,E1 0.577,E2 372.6037} C_DIS
LIN {X -6.6348,Y 141.9343,Z 192,A 82.2006,B 0.5556,C -0.0993,E1 0.5801,E2 373.6574} C_DIS
LIN {X -2.9354,Y 142.0593,Z 192,A 80.6856,B 0.5557,C -0.0982,E1 0.5845,E2 375.174} C_DIS
LIN {X 1.0853,Y 142.0847,Z 192,A 79.1897,B 0.5559,C -0.0972,E1 0.5888,E2 376.6573} C_DIS
LIN {X 4.9367,Y 142.004,Z 192,A 77.8921,B 0.5561,C -0.0963,E1 0.5925,E2 377.9301} C_DIS
LIN {X 7.9335,Y 141.869,Z 192,A 76.7465,B 0.5562,C -0.0954,E1 0.5958,E2 379.0692} C_DIS
LIN {X 10.9472,Y 141.6674,Z 192,A 75.6326,B 0.5564,C -0.0944,E1 0.5989,E2 380.1726} C_DIS
LIN {X 13.6992,Y 141.4265,Z 192,A 74.5514,B 0.5566,C -0.0934,E1 0.6021,E2 381.2503} C_DIS
LIN {X 17.5416,Y 141.0032,Z 192,A 73.1505,B 0.5568,C -0.092,E1 0.606,E2 382.6356} C_DIS
LIN {X 21.4687,Y 140.4573,Z 192,A 71.6395,B 0.5571,C -0.0904,E1 0.6103,E2 384.1375} C_DIS
LIN {X 25.9696,Y 139.6967,Z 192,A 70.1108,B 0.5573,C -0.0889,E1 0.6146,E2 385.6352} C_DIS
LIN {X 28.6089,Y 139.1786,Z 192,A 69.1432,B 0.5575,C -0.0878,E1 0.6173,E2 386.591} C_DIS
LIN {X 31.9935,Y 138.4399,Z 192,A 67.8286,B 0.5577,C -0.0862,E1 0.621,E2 387.8971} C_DIS
LIN {X 35.9496,Y 137.4668,Z 192,A 66.4443,B 0.558,C -0.0846,E1 0.6248,E2 389.2555} C_DIS
LIN {X 39.2082,Y 136.5734,Z 192,A 65.2188,B 0.5582,C -0.083,E1 0.6281,E2 390.467} C_DIS
LIN {X 43.831,Y 135.1601,Z 192,A 63.4798,B 0.5586,C -0.0807,E1 0.6329,E2 392.1846} C_DIS
LIN {X 47.2459,Y 134.0052,Z 192,A 62.2053,B 0.5588,C -0.0789,E1 0.6363,E2 393.4408} C_DIS
LIN {X 50.0481,Y 132.9821,Z 192,A 61.1883,B 0.559,C -0.0776,E1 0.639,E2 394.4386} C_DIS
LIN {X 52.8743,Y 131.8839,Z 192,A 60.1283,B 0.5592,C -0.076,E1 0.6418,E2 395.4818} C_DIS
LIN {X 55.6988,Y 130.718,Z 192,A 59.0449,B 0.5594,C -0.0744,E1 0.6446,E2 396.5499} C_DIS
LIN {X 58.4723,Y 129.4999,Z 192,A 57.9571,B 0.5597,C -0.0727,E1 0.6474,E2 397.6237} C_DIS
LIN {X 61.8083,Y 127.9417,Z 192,A 56.6569,B 0.5599,C -0.0706,E1 0.6507,E2 398.9047} C_DIS
LIN {X 65.7133,Y 125.9797,Z 192,A 55.1669,B 0.5602,C -0.0682,E1 0.6544,E2 400.3662} C_DIS
LIN {X 69.4027,Y 123.9874,Z 192,A 53.6271,B 0.5605,C -0.0655,E1 0.6583,E2 401.8901} C_DIS
LIN {X 73.6124,Y 121.5351,Z 192,A 51.9147,B 0.5609,C -0.0626,E1 0.6624,E2 403.5758} C_DIS
LIN {X 77.7326,Y 118.9427,Z 192,A 50.2802,B 0.5612,C -0.0597,E1 0.6662,E2 405.1754} C_DIS
LIN {X 81.5701,Y 116.3444,Z 192,A 48.7852,B 0.5615,C -0.0572,E1 0.6696,E2 406.6304} C_DIS
LIN {X 84.8555,Y 113.9697,Z 192,A 47.3421,B 0.5617,C -0.0544,E1 0.6729,E2 408.0528} C_DIS
LIN {X 88.5135,Y 111.1527,Z 192,A 45.8163,B 0.562,C -0.0516,E1 0.6762,E2 409.5422} C_DIS
LIN {X 91.6665,Y 108.5679,Z 192,A 44.4328,B 0.5622,C -0.0489,E1 0.6792,E2 410.8972} C_DIS
LIN {X 94.7241,Y 105.9098,Z 192,A 43.0731,B 0.5625,C -0.0463,E1 0.682,E2 412.2267} C_DIS
LIN {X 97.9237,Y 102.9593,Z 192,A 41.4826,B 0.5627,C -0.0429,E1 0.6853,E2 413.7991} C_DIS
LIN {X 101.7088,Y 99.222,Z 192,A 39.7821,B 0.563,C -0.0396,E1 0.6886,E2 415.4502} C_DIS
LIN {X 104.8681,Y 95.8769,Z 192,A 38.3024,B 0.5632,C -0.0366,E1 0.6914,E2 416.8877} C_DIS
LIN {X 107.5488,Y 92.8592,Z 192,A 36.9612,B 0.5633,C -0.0338,E1 0.6938,E2 418.1965} C_DIS
LIN {X 110.1474,Y 89.7615,Z 192,A 35.6236,B 0.5635,C -0.031,E1 0.6961,E2 419.5008} C_DIS
LIN {X 112.8748,Y 86.3066,Z 192,A 34.1756,B 0.5637,C -0.0279,E1 0.6986,E2 420.9113} C_DIS
LIN {X 115.3845,Y 82.9222,Z 192,A 32.7221,B 0.5638,C -0.0247,E1 0.7009,E2 422.3366} C_DIS
LIN {X 118.0066,Y 79.1461,Z 192,A 31.2108,B 0.564,C -0.0214,E1 0.7033,E2 423.8083} C_DIS
LIN {X 120.4879,Y 75.3146,Z 192,A 29.702,B 0.564,C -0.018,E1 0.7055,E2 425.2783} C_DIS
LIN {X 122.8774,Y 71.3493,Z 192,A 28.1893,B 0.5642,C -0.0147,E1 0.7076,E2 426.7493} C_DIS
LIN {X 125.001,Y 67.5605,Z 192,A 26.7387,B 0.5642,C -0.0114,E1 0.7095,E2 428.1644} C_DIS
LIN {X 126.9758,Y 63.7708,Z 192,A 25.4339,B 0.5642,C -0.0086,E1 0.7111,E2 429.4191} C_DIS
LIN {X 128.3589,Y 60.935,Z 192,A 24.3954,B 0.5643,C -0.0062,E1 0.7124,E2 430.4295} C_DIS
LIN {X 129.9846,Y 57.3886,Z 192,A 23.1358,B 0.5643,C -0.0033,E1 0.7138,E2 431.6513} C_DIS
LIN {X 131.2233,Y 54.4933,Z 192,A 22.1271,B 0.5643,C -0.001,E1 0.7148,E2 432.6282} C_DIS
LIN {X 132.3531,Y 51.6885,Z 192,A 21.0728,B 0.5643,C 0.0016,E1 0.7159,E2 433.6625} C_DIS
LIN {X 133.7758,Y 47.8868,Z 192,A 19.8079,B 0.5643,C 0.0044,E1 0.7171,E2 434.8818} C_DIS
LIN {X 134.9501,Y 44.4711,Z 192,A 18.6001,B 0.5643,C 0.0073,E1 0.7181,E2 436.059} C_DIS
LIN {X 136.5513,Y 39.2838,Z 192,A 16.8137,B 0.5643,C 0.0115,E1 0.7195,E2 437.7955} C_DIS
LIN {X 137.3527,Y 36.3777,Z 192,A 15.8638,B 0.5642,C 0.0137,E1 0.7202,E2 438.7122} C_DIS
LIN {X 138.2524,Y 32.7961,Z 192,A 14.6641,B 0.5642,C 0.0165,E1 0.721,E2 439.8756} C_DIS
LIN {X 139.1551,Y 28.7243,Z 192,A 13.1917,B 0.564,C 0.0203,E1 0.7218,E2 441.3219} C_DIS
LIN {X 140.1997,Y 23.0913,Z 192,A 11.38,B 0.5638,C 0.0245,E1 0.7227,E2 443.0703} C_DIS
LIN {X 140.776,Y 19.2843,Z 192,A 10.2197,B 0.5638,C 0.0271,E1 0.7231,E2 444.1803} C_DIS
LIN {X 141.1377,Y 16.4143,Z 192,A 9.2951,B 0.5636,C 0.0293,E1 0.7234,E2 445.0737} C_DIS
LIN {X 141.4413,Y 13.5454,Z 192,A 8.3296,B 0.5635,C 0.0316,E1 0.7237,E2 446.0137} C_DIS
LIN {X 141.7394,Y 9.9603,Z 192,A 7.1745,B 0.5633,C 0.0343,E1 0.7239,E2 447.1305} C_DIS
LIN {X 141.9294,Y 6.7325,Z 192,A 6.1416,B 0.5632,C 0.0368,E1 0.7241,E2 448.1282} C_DIS
LIN {X 142.0393,Y 3.7438,Z 192,A 5.1751,B 0.563,C 0.0391,E1 0.7241,E2 449.0633} C_DIS
LIN {X 142.0919,Y 0.0438,Z 192,A 3.7977,B 0.5627,C 0.0427,E1 0.7241,E2 450.4263} C_DIS
LIN {X 142.0268,Y -4.1951,Z 192,A 2.5792,B 0.5625,C 0.0453,E1 0.7241,E2 451.5796} C_DIS
LIN {X 141.8937,Y -7.4432,Z 192,A 1.5458,B 0.5623,C 0.0477,E1 0.724,E2 452.5761} C_DIS
LIN {X 141.7081,Y -10.389,Z 192,A 0.5223,B 0.5621,C 0.0503,E1 0.7238,E2 453.5775} C_DIS
LIN {X 141.3055,Y -14.8976,Z 192,A -0.8847,B 0.5618,C 0.0535,E1 0.7234,E2 454.9284} C_DIS
LIN {X 140.9565,Y -17.9076,Z 192,A -1.8173,B 0.5616,C 0.0556,E1 0.7231,E2 455.8221} C_DIS
LIN {X 140.4213,Y -21.7014,Z 192,A -3.0869,B 0.5613,C 0.0586,E1 0.7226,E2 457.0545} C_DIS
LIN {X 139.9767,Y -24.4131,Z 192,A -3.9748,B 0.5611,C 0.0607,E1 0.7222,E2 457.9126} C_DIS
LIN {X 139.4789,Y -27.1088,Z 192,A -4.9019,B 0.5608,C 0.0629,E1 0.7218,E2 458.8156} C_DIS
LIN {X 138.9231,Y -29.8237,Z 192,A -5.7734,B 0.5606,C 0.0649,E1 0.7213,E2 459.6533} C_DIS
LIN {X 138.3017,Y -32.5917,Z 192,A -6.8446,B 0.5603,C 0.0677,E1 0.7206,E2 460.7152} C_DIS
LIN {X 137.0699,Y -37.4377,Z 192,A -8.3823,B 0.5599,C 0.0711,E1 0.7196,E2 462.1869} C_DIS
LIN {X 134.6954,Y -45.2359,Z 192,A -11.0397,B 0.5591,C 0.0771,E1 0.7175,E2 464.7571} C_DIS
LIN {X 133.7017,Y -48.0923,Z 192,A -12.004,B 0.5588,C 0.0793,E1 0.7166,E2 465.6857} C_DIS
LIN {X 132.6045,Y -51.0419,Z 192,A -13.0208,B 0.5584,C 0.0815,E1 0.7156,E2 466.6673} C_DIS
LIN {X 131.4413,Y -53.9712,Z 192,A -14.2535,B 0.558,C 0.0847,E1 0.7143,E2 467.8955} C_DIS
LIN {X 129.6162,Y -58.2124,Z 192,A -15.574,B 0.5576,C 0.0873,E1 0.7129,E2 469.1391} C_DIS
LIN {X 127.614,Y -62.4805,Z 192,A -17.0443,B 0.5571,C 0.0904,E1 0.7112,E2 470.5482} C_DIS
LIN {X 125.8275,Y -66.0031,Z 192,A -18.4846,B 0.5565,C 0.0938,E1 0.7094,E2 471.9674} C_DIS
LIN {X 123.7848,Y -69.7632,Z 192,A -20.1682,B 0.5558,C 0.098,E1 0.7071,E2 473.6462} C_DIS
LIN {X 121.8667,Y -73.0624,Z 192,A -21.2841,B 0.5554,C 0.1001,E1 0.7056,E2 474.7012} C_DIS
LIN {X 119.5864,Y -76.7377,Z 192,A -22.6237,B 0.5549,C 0.1028,E1 0.7037,E2 475.9825} C_DIS
LIN {X 117.1525,Y -80.4042,Z 192,A -24.0849,B 0.5544,C 0.1058,E1 0.7014,E2 477.3986} C_DIS
LIN {X 114.5647,Y -84.0505,Z 192,A -25.5827,B 0.5537,C 0.1089,E1 0.699,E2 478.8524} C_DIS
LIN {X 111.7376,Y -87.7739,Z 192,A -27.1456,B 0.5531,C 0.1121,E1 0.6964,E2 480.3686} C_DIS
LIN {X 108.8081,Y -91.3803,Z 192,A -28.6914,B 0.5525,C 0.1152,E1 0.6937,E2 481.8666} C_DIS
LIN {X 105.8942,Y -94.7416,Z 192,A -30.1883,B 0.5518,C 0.1182,E1 0.691,E2 483.3202} C_DIS
LIN {X 102.7306,Y -98.163,Z 192,A -31.7663,B 0.5512,C 0.1213,E1 0.688,E2 484.8541} C_DIS
LIN {X 99.3688,Y -101.5649,Z 192,A -33.3745,B 0.5505,C 0.1243,E1 0.6849,E2 486.4153} C_DIS
LIN {X 95.8973,Y -104.8493,Z 192,A -34.9839,B 0.5498,C 0.1273,E1 0.6817,E2 487.9777} C_DIS
LIN {X 92.4034,Y -107.9414,Z 192,A -36.5704,B 0.5491,C 0.1302,E1 0.6784,E2 489.5206} C_DIS
LIN {X 88.8496,Y -110.8851,Z 192,A -38.1489,B 0.5485,C 0.1331,E1 0.675,E2 491.0573} C_DIS
LIN {X 85.1231,Y -113.7705,Z 192,A -39.663,B 0.5479,C 0.1355,E1 0.6717,E2 492.5134} C_DIS
LIN {X 81.7332,Y -116.2294,Z 192,A -41.1604,B 0.5472,C 0.1382,E1 0.6683,E2 493.9825} C_DIS
LIN {X 78.0285,Y -118.7481,Z 192,A -42.6914,B 0.5465,C 0.1407,E1 0.6648,E2 495.4723} C_DIS
LIN {X 74.2729,Y -121.1325,Z 192,A -44.2199,B 0.5459,C 0.1432,E1 0.6612,E2 496.961} C_DIS
LIN {X 70.414,Y -123.4156,Z 192,A -45.7444,B 0.5453,C 0.1455,E1 0.6575,E2 498.4427} C_DIS
LIN {X 65.9465,Y -125.8572,Z 192,A -47.5198,B 0.5445,C 0.1482,E1 0.6532,E2 500.1762} C_DIS
LIN {X 62.7115,Y -127.5001,Z 192,A -48.792,B 0.544,C 0.1501,E1 0.65,E2 501.4198} C_DIS
LIN {X 58.526,Y -129.4759,Z 192,A -50.666,B 0.5431,C 0.1533,E1 0.6451,E2 503.2964} C_DIS
LIN {X 55.1289,Y -130.9578,Z 192,A -51.7654,B 0.5428,C 0.1544,E1 0.6423,E2 504.3348} C_DIS
LIN {X 51.3558,Y -132.4825,Z 192,A -53.1081,B 0.5424,C 0.1561,E1 0.6389,E2 505.6317} C_DIS
LIN {X 48.212,Y -133.6585,Z 192,A -54.3068,B 0.5419,C 0.1576,E1 0.6357,E2 506.8069} C_DIS
LIN {X 44.796,Y -134.8419,Z 192,A -55.9048,B 0.5411,C 0.1603,E1 0.6313,E2 508.4283} C_DIS
LIN {X 41.0293,Y -136.0366,Z 192,A -56.9845,B 0.5409,C 0.1609,E1 0.6285,E2 509.4279} C_DIS
LIN {X 37.4172,Y -137.0755,Z 192,A -58.3325,B 0.5405,C 0.1625,E1 0.6249,E2 510.7504} C_DIS
LIN {X 34.2236,Y -137.907,Z 192,A -59.6153,B 0.54,C 0.1641,E1 0.6213,E2 512.0266} C_DIS
LIN {X 28.517,Y -139.1973,Z 192,A -61.7836,B 0.5392,C 0.1665,E1 0.6153,E2 514.1661} C_DIS
LIN {X 24.3035,Y -139.9963,Z 192,A -63.1971,B 0.5389,C 0.1677,E1 0.6114,E2 515.5304} C_DIS
LIN {X 21.4505,Y -140.4601,Z 192,A -64.2344,B 0.5386,C 0.1686,E1 0.6085,E2 516.548} C_DIS
LIN {X 18.5682,Y -140.8699,Z 192,A -65.2919,B 0.5383,C 0.1696,E1 0.6055,E2 517.5877} C_DIS
LIN {X 15.2394,Y -141.2688,Z 192,A -66.6103,B 0.5379,C 0.1709,E1 0.6017,E2 518.9017} C_DIS
LIN {X 11.1597,Y -141.6517,Z 192,A -68.2254,B 0.5374,C 0.1724,E1 0.5971,E2 520.512} C_DIS
LIN {X 7.2812,Y -141.9018,Z 192,A -69.5075,B 0.5372,C 0.1731,E1 0.5935,E2 521.7492} C_DIS
LIN {X 4.241,Y -142.0255,Z 192,A -70.6579,B 0.5369,C 0.1739,E1 0.5902,E2 522.8881} C_DIS
LIN {X 1.0199,Y -142.0827,Z 192,A -71.4225,B 0.5369,C 0.1737,E1 0.5882,E2 523.5674} C_DIS
Enddeposition()
LIN {X 1.0199,Y -142.0827,Z 192,A -71.4228,B 0.5369,C 0.1737,E1 0.5882,E2 523.5677} C_DIS
Startdeposition()
$VEL.CP = VEL_PRINT
LIN {X 1.7649,Y -142.9779,Z 192,A -71.0319,B 0.5371,C 0.1734,E1 0.5894,E2 523.179} C_DIS
LIN {X 5.2703,Y -142.8906,Z 192,A -69.7359,B 0.5374,C 0.1725,E1 0.5931,E2 521.8998} C_DIS
LIN {X 8.7718,Y -142.718,Z 192,A -68.4428,B 0.5377,C 0.1715,E1 0.5968,E2 520.6239} C_DIS
LIN {X 12.2877,Y -142.4586,Z 192,A -67.1475,B 0.538,C 0.1705,E1 0.6005,E2 519.3469} C_DIS
LIN {X 15.7763,Y -142.1151,Z 192,A -65.8636,B 0.5384,C 0.1694,E1 0.6041,E2 518.0816} C_DIS
LIN {X 19.2534,Y -141.6867,Z 192,A -64.5846,B 0.5387,C 0.1682,E1 0.6077,E2 516.8219} C_DIS
LIN {X 22.7196,Y -141.173,Z 192,A -63.2884,B 0.5391,C 0.1669,E1 0.6114,E2 515.5422} C_DIS
LIN {X 26.2217,Y -140.5637,Z 192,A -62.0039,B 0.5395,C 0.1657,E1 0.615,E2 514.2793} C_DIS
LIN {X 29.6572,Y -139.8787,Z 192,A -60.7429,B 0.5399,C 0.1644,E1 0.6185,E2 513.0403} C_DIS
LIN {X 33.0686,Y -139.1114,Z 192,A -59.4887,B 0.5403,C 0.163,E1 0.6219,E2 511.8089} C_DIS
LIN {X 36.4549,Y -138.2624,Z 192,A -58.1337,B 0.5409,C 0.1613,E1 0.6257,E2 510.4599} C_DIS
LIN {X 39.8169,Y -137.3319,Z 192,A -56.9977,B 0.5412,C 0.1601,E1 0.6287,E2 509.3651} C_DIS
LIN {X 43.1581,Y -136.3187,Z 192,A -55.7504,B 0.5416,C 0.1586,E1 0.6321,E2 508.1411} C_DIS
LIN {X 46.521,Y -135.2079,Z 192,A -54.5059,B 0.5421,C 0.157,E1 0.6354,E2 506.9236} C_DIS
LIN {X 49.8219,Y -134.0267,Z 192,A -53.1845,B 0.5426,C 0.1552,E1 0.6389,E2 505.6145} C_DIS
LIN {X 54.3264,Y -132.2672,Z 192,A -51.4691,B 0.5433,C 0.1528,E1 0.6434,E2 503.9333} C_DIS
LIN {X 57.9712,Y -130.7088,Z 192,A -50.1926,B 0.5437,C 0.1512,E1 0.6466,E2 502.7053} C_DIS
LIN {X 61.1499,Y -129.2525,Z 192,A -48.9771,B 0.5442,C 0.1495,E1 0.6497,E2 501.5183} C_DIS
LIN {X 64.6033,Y -127.5607,Z 192,A -47.7323,B 0.5447,C 0.1478,E1 0.6528,E2 500.3194} C_DIS
LIN {X 68.0036,Y -125.7834,Z 192,A -46.2817,B 0.5453,C 0.1454,E1 0.6564,E2 498.8814} C_DIS
LIN {X 71.2487,Y -123.9744,Z 192,A -45.0281,B 0.5458,C 0.1435,E1 0.6595,E2 497.6638} C_DIS
LIN {X 74.2672,Y -122.1896,Z 192,A -43.78,B 0.5464,C 0.1414,E1 0.6625,E2 496.4394} C_DIS
LIN {X 77.9747,Y -119.8573,Z 192,A -42.3273,B 0.547,C 0.1391,E1 0.6658,E2 495.033} C_DIS
LIN {X 80.8898,Y -117.9095,Z 192,A -41.1335,B 0.5475,C 0.1372,E1 0.6686,E2 493.8713} C_DIS
LIN {X 83.7693,Y -115.8816,Z 192,A -39.9374,B 0.548,C 0.1351,E1 0.6713,E2 492.7078} C_DIS
LIN {X 86.8292,Y -113.6068,Z 192,A -38.5706,B 0.5486,C 0.1326,E1 0.6743,E2 491.3651} C_DIS
LIN {X 90.0324,Y -111.086,Z 192,A -37.2571,B 0.5491,C 0.1304,E1 0.6771,E2 490.1002} C_DIS
LIN {X 92.7279,Y -108.8456,Z 192,A -36.0772,B 0.5496,C 0.1283,E1 0.6796,E2 488.9542} C_DIS
LIN {X 95.3796,Y -106.5295,Z 192,A -34.8254,B 0.5502,C 0.1259,E1 0.6822,E2 487.7259} C_DIS
LIN {X 98.6002,Y -103.5562,Z 192,A -33.4277,B 0.5507,C 0.1234,E1 0.685,E2 486.3824} C_DIS
LIN {X 101.11,Y -101.1078,Z 192,A -32.243,B 0.5512,C 0.1212,E1 0.6873,E2 485.2306} C_DIS
LIN {X 103.5579,Y -98.5984,Z 192,A -31.0742,B 0.5517,C 0.1189,E1 0.6895,E2 484.097} C_DIS
LIN {X 105.9535,Y -96.0192,Z 192,A -29.9033,B 0.5522,C 0.1167,E1 0.6917,E2 482.9618} C_DIS
LIN {X 108.2763,Y -93.392,Z 192,A -28.7397,B 0.5527,C 0.1144,E1 0.6938,E2 481.8341} C_DIS
LIN {X 110.5331,Y -90.7102,Z 192,A -27.5785,B 0.5531,C 0.1121,E1 0.6958,E2 480.709} C_DIS
LIN {X 112.725,Y -87.972,Z 192,A -26.39,B 0.5536,C 0.1096,E1 0.6979,E2 479.5524} C_DIS
LIN {X 115.3773,Y -84.4627,Z 192,A -24.8707,B 0.5543,C 0.1063,E1 0.7004,E2 478.0686} C_DIS
LIN {X 117.9112,Y -80.8873,Z 192,A -23.5105,B 0.5548,C 0.1037,E1 0.7025,E2 476.7669} C_DIS
LIN {X 119.8581,Y -77.9734,Z 192,A -22.2536,B 0.5553,C 0.1008,E1 0.7044,E2 475.5311} C_DIS
LIN {X 122.2159,Y -74.2238,Z 192,A -20.9037,B 0.5558,C 0.0982,E1 0.7063,E2 474.2437} C_DIS
LIN {X 123.9951,Y -71.2123,Z 192,A -19.7526,B 0.5562,C 0.0957,E1 0.7078,E2 473.129} C_DIS
LIN {X 125.699,Y -68.1594,Z 192,A -18.5513,B 0.5567,C 0.093,E1 0.7094,E2 471.9563} C_DIS
LIN {X 127.3245,Y -65.0673,Z 192,A -17.4666,B 0.557,C 0.0908,E1 0.7108,E2 470.9173} C_DIS
LIN {X 128.8737,Y -61.9429,Z 192,A -16.32,B 0.5574,C 0.0883,E1 0.7121,E2 469.8068} C_DIS
LIN {X 130.3637,Y -58.7428,Z 192,A -15.3024,B 0.5577,C 0.0863,E1 0.7133,E2 468.8466} C_DIS
LIN {X 131.4212,Y -56.3374,Z 192,A -14.3106,B 0.5581,C 0.0838,E1 0.7144,E2 467.863} C_DIS
LIN {X 132.7659,Y -53.0907,Z 192,A -13.167,B 0.5585,C 0.0812,E1 0.7155,E2 466.7571} C_DIS
LIN {X 134.0283,Y -49.8178,Z 192,A -12.0263,B 0.5589,C 0.0787,E1 0.7166,E2 465.654} C_DIS
LIN {X 135.2119,Y -46.5093,Z 192,A -10.8781,B 0.5592,C 0.076,E1 0.7177,E2 464.5426} C_DIS
LIN {X 136.331,Y -43.1196,Z 192,A -9.6622,B 0.5596,C 0.0731,E1 0.7187,E2 463.3568} C_DIS
LIN {X 137.6165,Y -38.8214,Z 192,A -8.4204,B 0.5599,C 0.0708,E1 0.7196,E2 462.1937} C_DIS
LIN {X 138.272,Y -36.4188,Z 192,A -7.4653,B 0.5602,C 0.0682,E1 0.7203,E2 461.2441} C_DIS
LIN {X 139.1229,Y -33.0208,Z 192,A -6.3299,B 0.5606,C 0.0656,E1 0.721,E2 460.1462} C_DIS
LIN {X 139.8903,Y -29.6035,Z 192,A -5.198,B 0.5609,C 0.063,E1 0.7217,E2 459.052} C_DIS
LIN {X 140.6064,Y -25.9967,Z 192,A -4.0181,B 0.5612,C 0.0603,E1 0.7223,E2 457.9127} C_DIS
LIN {X 141.1735,Y -22.717,Z 192,A -2.9206,B 0.5614,C 0.0576,E1 0.7227,E2 456.8478} C_DIS
LIN {X 141.6894,Y -19.2327,Z 192,A -1.7789,B 0.5617,C 0.0549,E1 0.7232,E2 455.743} C_DIS
LIN {X 142.1178,Y -15.751,Z 192,A -0.6479,B 0.562,C 0.0523,E1 0.7235,E2 454.6496} C_DIS
LIN {X 142.4605,Y -12.2653,Z 192,A 0.4797,B 0.5622,C 0.0496,E1 0.7238,E2 453.5595} C_DIS
LIN {X 142.7183,Y -8.7678,Z 192,A 1.6061,B 0.5624,C 0.047,E1 0.724,E2 452.4709} C_DIS
LIN {X 142.8906,Y -5.2695,Z 192,A 2.7425,B 0.5626,C 0.0443,E1 0.7241,E2 451.3705} C_DIS
LIN {X 142.978,Y -1.7534,Z 192,A 3.824,B 0.5628,C 0.0418,E1 0.7241,E2 450.3332} C_DIS
LIN {X 142.9667,Y 2.4367,Z 192,A 5.1082,B 0.563,C 0.0389,E1 0.7241,E2 449.102} C_DIS
LIN {X 142.8908,Y 5.265,Z 192,A 6.1445,B 0.5632,C 0.0362,E1 0.7241,E2 448.0783} C_DIS
LIN {X 142.7184,Y 8.7652,Z 192,A 7.2985,B 0.5634,C 0.0334,E1 0.7239,E2 446.9574} C_DIS
LIN {X 142.4591,Y 12.2818,Z 192,A 8.4022,B 0.5635,C 0.0308,E1 0.7237,E2 445.8946} C_DIS
LIN {X 142.1158,Y 15.7697,Z 192,A 9.5301,B 0.5637,C 0.0282,E1 0.7233,E2 444.8031} C_DIS
LIN {X 141.6875,Y 19.2469,Z 192,A 10.6592,B 0.5638,C 0.0255,E1 0.723,E2 443.7099} C_DIS
LIN {X 141.174,Y 22.7135,Z 192,A 11.8193,B 0.5639,C 0.0227,E1 0.7225,E2 442.5816} C_DIS
LIN {X 140.5668,Y 26.2056,Z 192,A 12.9502,B 0.564,C 0.02,E1 0.7219,E2 441.4882} C_DIS
LIN {X 139.883,Y 29.6373,Z 192,A 14.0782,B 0.5641,C 0.0173,E1 0.7213,E2 440.3956} C_DIS
LIN {X 139.0239,Y 33.4317,Z 192,A 15.2575,B 0.5641,C 0.0147,E1 0.7206,E2 439.265} C_DIS
LIN {X 138.2677,Y 36.4352,Z 192,A 16.3347,B 0.5643,C 0.012,E1 0.7199,E2 438.2086} C_DIS
LIN {X 137.3362,Y 39.802,Z 192,A 17.5307,B 0.5643,C 0.0091,E1 0.719,E2 437.0384} C_DIS
LIN {X 136.3101,Y 43.1852,Z 192,A 18.6082,B 0.5643,C 0.0067,E1 0.7181,E2 436.0038} C_DIS
LIN {X 134.9455,Y 47.2778,Z 192,A 19.9108,B 0.5643,C 0.0038,E1 0.717,E2 434.755} C_DIS
LIN {X 134.0247,Y 49.8273,Z 192,A 20.884,B 0.5643,C 0.0014,E1 0.7161,E2 433.7957} C_DIS
LIN {X 132.7627,Y 53.0987,Z 192,A 22.0203,B 0.5643,C -0.0013,E1 0.7149,E2 432.693} C_DIS
LIN {X 131.4222,Y 56.3351,Z 192,A 23.1604,B 0.5643,C -0.0039,E1 0.7137,E2 431.5855} C_DIS
LIN {X 129.997,Y 59.5506,Z 192,A 24.3337,B 0.5643,C -0.0066,E1 0.7124,E2 430.4413} C_DIS
LIN {X 128.5005,Y 62.7153,Z 192,A 25.4361,B 0.5643,C -0.0091,E1 0.7111,E2 429.3758} C_DIS
LIN {X 126.9275,Y 65.8418,Z 192,A 26.6651,B 0.5643,C -0.012,E1 0.7096,E2 428.1679} C_DIS
LIN {X 124.8398,Y 69.7207,Z 192,A 28.0148,B 0.5642,C -0.0149,E1 0.7078,E2 426.8688} C_DIS
LIN {X 123.0931,Y 72.7602,Z 192,A 29.1679,B 0.5642,C -0.0175,E1 0.7062,E2 425.746} C_DIS
LIN {X 121.2718,Y 75.7564,Z 192,A 30.3131,B 0.564,C -0.02,E1 0.7046,E2 424.6319} C_DIS
LIN {X 119.3781,Y 78.7064,Z 192,A 31.4594,B 0.564,C -0.0225,E1 0.7029,E2 423.5165} C_DIS
LIN {X 117.4123,Y 81.6099,Z 192,A 32.6072,B 0.5638,C -0.025,E1 0.7011,E2 422.3993} C_DIS
LIN {X 114.9603,Y 85.0303,Z 192,A 34.0473,B 0.5637,C -0.0283,E1 0.6987,E2 420.9882} C_DIS
LIN {X 112.7166,Y 87.9828,Z 192,A 35.2148,B 0.5635,C -0.0307,E1 0.6968,E2 419.8582} C_DIS
LIN {X 110.5268,Y 90.7178,Z 192,A 36.3869,B 0.5635,C -0.0332,E1 0.6947,E2 418.7131} C_DIS
LIN {X 107.6981,Y 94.0581,Z 192,A 37.8145,B 0.5632,C -0.0361,E1 0.6922,E2 417.3234} C_DIS
LIN {X 104.9301,Y 97.1373,Z 192,A 39.2306,B 0.563,C -0.0391,E1 0.6895,E2 415.9354} C_DIS
LIN {X 102.3402,Y 99.862,Z 192,A 40.5367,B 0.5628,C -0.0419,E1 0.687,E2 414.6522} C_DIS
LIN {X 99.2193,Y 102.9633,Z 192,A 41.9027,B 0.5626,C -0.0444,E1 0.6844,E2 413.3316} C_DIS
LIN {X 96.5246,Y 105.4937,Z 192,A 43.238,B 0.5624,C -0.0472,E1 0.6816,E2 412.0128} C_DIS
LIN {X 93.1281,Y 108.5036,Z 192,A 44.7262,B 0.5622,C -0.0501,E1 0.6785,E2 410.5619} C_DIS
LIN {X 90.0362,Y 111.0829,Z 192,A 45.9941,B 0.5619,C -0.0524,E1 0.6758,E2 409.3327} C_DIS
LIN {X 87.2877,Y 113.2555,Z 192,A 47.2148,B 0.5617,C -0.0547,E1 0.6731,E2 408.1324} C_DIS
LIN {X 83.7538,Y 115.8928,Z 192,A 48.6695,B 0.5615,C -0.0573,E1 0.6699,E2 406.7123} C_DIS
LIN {X 80.886,Y 117.9122,Z 192,A 49.854,B 0.5612,C -0.0595,E1 0.6671,E2 405.5521} C_DIS
LIN {X 77.9707,Y 119.86,Z 192,A 51.1103,B 0.561,C -0.0618,E1 0.6642,E2 404.3121} C_DIS
LIN {X 74.5212,Y 122.0348,Z 192,A 52.4568,B 0.5607,C -0.064,E1 0.661,E2 402.997} C_DIS
LIN {X 71.2434,Y 123.9774,Z 192,A 53.738,B 0.5605,C -0.0662,E1 0.6579,E2 401.7424} C_DIS
LIN {X 68.1826,Y 125.6864,Z 192,A 55.0198,B 0.5602,C -0.0684,E1 0.6547,E2 400.474} C_DIS
LIN {X 65.0582,Y 127.3291,Z 192,A 56.1457,B 0.56,C -0.0701,E1 0.6519,E2 399.3789} C_DIS
LIN {X 61.9226,Y 128.8834,Z 192,A 57.3851,B 0.5598,C -0.0721,E1 0.6488,E2 398.157} C_DIS
LIN {X 58.7384,Y 130.3656,Z 192,A 58.6441,B 0.5595,C -0.0741,E1 0.6456,E2 396.9139} C_DIS
LIN {X 54.7181,Y 132.1036,Z 192,A 60.0954,B 0.5592,C -0.0762,E1 0.6418,E2 395.4948} C_DIS
LIN {X 51.461,Y 133.406,Z 192,A 61.3185,B 0.559,C -0.078,E1 0.6386,E2 394.2909} C_DIS
LIN {X 48.1626,Y 134.6319,Z 192,A 62.6709,B 0.5587,C -0.08,E1 0.635,E2 392.9449} C_DIS
LIN {X 44.8124,Y 135.7839,Z 192,A 63.7952,B 0.5585,C -0.0814,E1 0.632,E2 391.8514} C_DIS
LIN {X 41.4738,Y 136.8406,Z 192,A 65.0298,B 0.5582,C -0.083,E1 0.6286,E2 390.6344} C_DIS
LIN {X 38.1152,Y 137.814,Z 192,A 66.2683,B 0.558,C -0.0846,E1 0.6252,E2 389.4129} C_DIS
LIN {X 34.6606,Y 138.7236,Z 192,A 67.5333,B 0.5578,C -0.0861,E1 0.6218,E2 388.1652} C_DIS
LIN {X 31.3155,Y 139.5168,Z 192,A 68.7657,B 0.5575,C -0.0876,E1 0.6183,E2 386.9478} C_DIS
LIN {X 27.8898,Y 140.2422,Z 192,A 70.0206,B 0.5573,C -0.089,E1 0.6148,E2 385.7082} C_DIS
LIN {X 24.4373,Y 140.8855,Z 192,A 71.3956,B 0.5571,C -0.0906,E1 0.6109,E2 384.3369} C_DIS
LIN {X 20.9772,Y 141.4421,Z 192,A 72.5748,B 0.5569,C -0.0917,E1 0.6076,E2 383.1806} C_DIS
LIN {X 17.5047,Y 141.9129,Z 192,A 73.9235,B 0.5566,C -0.0931,E1 0.6038,E2 381.8378} C_DIS
LIN {X 13.9978,Y 142.3009,Z 192,A 75.1337,B 0.5565,C -0.0942,E1 0.6003,E2 380.6482} C_DIS
LIN {X 10.5082,Y 142.6007,Z 192,A 76.4162,B 0.5563,C -0.0953,E1 0.5967,E2 379.3782} C_DIS
LIN {X 7.0105,Y 142.8155,Z 192,A 77.7028,B 0.5561,C -0.0963,E1 0.593,E2 378.1036} C_DIS
LIN {X 3.5085,Y 142.9451,Z 192,A 78.9939,B 0.5559,C -0.0973,E1 0.5893,E2 376.8241} C_DIS
LIN {X -0.0059,Y 142.9896,Z 192,A 80.3449,B 0.5557,C -0.0983,E1 0.5854,E2 375.4792} C_DIS
LIN {X -3.5235,Y 142.9447,Z 192,A 81.727,B 0.5556,C -0.0993,E1 0.5814,E2 374.1003} C_DIS
LIN {X -7.0245,Y 142.8148,Z 192,A 82.9674,B 0.5555,C -0.1,E1 0.5778,E2 372.8763} C_DIS
LIN {X -10.524,Y 142.5996,Z 192,A 84.2902,B 0.5553,C -0.1007,E1 0.574,E2 371.562} C_DIS
LIN {X -14.4279,Y 142.2596,Z 192,A 85.7678,B 0.5553,C -0.1014,E1 0.5698,E2 370.0941} C_DIS
LIN {X -17.5259,Y 141.9104,Z 192,A 86.9749,B 0.5551,C -0.1019,E1 0.5663,E2 368.8915} C_DIS
LIN {X -20.9935,Y 141.4398,Z 192,A 88.3321,B 0.5551,C -0.1024,E1 0.5624,E2 367.5392} C_DIS
LIN {X -24.4537,Y 140.8826,Z 192,A 89.708,B 0.5549,C -0.1029,E1 0.5584,E2 366.1667} C_DIS
LIN {X -28.1332,Y 140.1927,Z 192,A 91.2391,B 0.5549,C -0.1033,E1 0.5541,E2 364.6331} C_DIS
LIN {X -33.1509,Y 139.0915,Z 192,A 93.1309,B 0.5549,C -0.1035,E1 0.5487,E2 362.7582} C_DIS
LIN {X -36.4256,Y 138.2702,Z 192,A 94.53,B 0.5548,C -0.1037,E1 0.5448,E2 361.3553} C_DIS
LIN {X -40.5941,Y 137.1043,Z 192,A 96.1312,B 0.5548,C -0.1036,E1 0.5403,E2 359.7676} C_DIS
LIN {X -43.2003,Y 136.3052,Z 192,A 97.3558,B 0.5548,C -0.1036,E1 0.5369,E2 358.5308} C_DIS
LIN {X -46.5264,Y 135.206,Z 192,A 98.7741,B 0.5548,C -0.1035,E1 0.533,E2 357.1117} C_DIS
LIN {X -49.8252,Y 134.0255,Z 192,A 100.2028,B 0.5548,C -0.1032,E1 0.5291,E2 355.6813} C_DIS
LIN {X -53.0956,Y 132.7639,Z 192,A 101.646,B 0.5549,C -0.1029,E1 0.5251,E2 354.2351} C_DIS
LIN {X -56.3475,Y 131.4169,Z 192,A 103.1021,B 0.555,C -0.1025,E1 0.5212,E2 352.7752} C_DIS
LIN {X -59.5669,Y 129.9895,Z 192,A 104.4243,B 0.5551,C -0.1019,E1 0.5178,E2 351.4623} C_DIS
LIN {X -62.8566,Y 128.4308,Z 192,A 106.123,B 0.5552,C -0.1013,E1 0.5132,E2 349.7411} C_DIS
LIN {X -65.8373,Y 126.9299,Z 192,A 107.4944,B 0.5554,C -0.1006,E1 0.5097,E2 348.3671} C_DIS
LIN {X -68.9669,Y 125.2578,Z 192,A 109.0071,B 0.5555,C -0.0997,E1 0.5058,E2 346.8463} C_DIS
LIN {X -72.0149,Y 123.5308,Z 192,A 110.521,B 0.5557,C -0.0988,E1 0.502,E2 345.3225} C_DIS
LIN {X -75.0204,Y 121.7285,Z 192,A 112.0327,B 0.5559,C -0.0977,E1 0.4982,E2 343.801} C_DIS
LIN {X -78.2894,Y 119.6526,Z 192,A 113.83,B 0.5561,C -0.0964,E1 0.4937,E2 341.9804} C_DIS
LIN {X -81.6106,Y 117.4118,Z 192,A 115.4767,B 0.5563,C -0.0949,E1 0.4898,E2 340.3304} C_DIS
LIN {X -84.482,Y 115.3632,Z 192,A 117.0298,B 0.5566,C -0.0935,E1 0.4861,E2 338.7643} C_DIS
LIN {X -87.2833,Y 113.259,Z 192,A 118.7288,B 0.5569,C -0.0919,E1 0.4822,E2 337.0367} C_DIS
LIN {X -90.7127,Y 110.531,Z 192,A 120.5749,B 0.5572,C -0.0898,E1 0.478,E2 335.1825} C_DIS
LIN {X -93.3933,Y 108.2752,Z 192,A 122.1777,B 0.5575,C -0.088,E1 0.4744,E2 333.5605} C_DIS
LIN {X -96.0342,Y 105.9399,Z 192,A 123.7687,B 0.5578,C -0.0861,E1 0.471,E2 331.9523} C_DIS
LIN {X -98.6021,Y 103.5543,Z 192,A 125.3788,B 0.5581,C -0.084,E1 0.4675,E2 330.3221} C_DIS
LIN {X -101.111,Y 101.1068,Z 192,A 127.0225,B 0.5584,C -0.0818,E1 0.4641,E2 328.6547} C_DIS
LIN {X -103.5579,Y 98.5984,Z 192,A 128.7188,B 0.5588,C -0.0795,E1 0.4607,E2 326.9291} C_DIS
LIN {X -106.5439,Y 95.3635,Z 192,A 130.7302,B 0.5592,C -0.0765,E1 0.4567,E2 324.893} C_DIS
LIN {X -108.8495,Y 92.7233,Z 192,A 132.3927,B 0.5595,C -0.0739,E1 0.4536,E2 323.2044} C_DIS
LIN {X -111.0891,Y 90.0285,Z 192,A 134.0677,B 0.5599,C -0.0713,E1 0.4505,E2 321.5017} C_DIS
LIN {X -113.6582,Y 86.7619,Z 192,A 136.1344,B 0.5603,C -0.0678,E1 0.4468,E2 319.3934} C_DIS
LIN {X -115.9022,Y 83.7409,Z 192,A 137.9208,B 0.5607,C -0.0647,E1 0.4437,E2 317.578} C_DIS
LIN {X -117.9172,Y 80.8786,Z 192,A 139.7593,B 0.561,C -0.0615,E1 0.4407,E2 315.6933} C_DIS
LIN {X -120.3352,Y 77.2352,Z 192,A 141.7914,B 0.5614,C -0.0576,E1 0.4374,E2 313.6316} C_DIS
LIN {X -122.1888,Y 74.2685,Z 192,A 143.5321,B 0.5618,C -0.0543,E1 0.4348,E2 311.8545} C_DIS
LIN {X -123.9703,Y 71.2558,Z 192,A 145.3015,B 0.5621,C -0.0508,E1 0.4322,E2 310.0453} C_DIS
LIN {X -125.6885,Y 68.1786,Z 192,A 147.1627,B 0.5624,C -0.0471,E1 0.4296,E2 308.1346} C_DIS
LIN {X -127.3241,Y 65.068,Z 192,A 148.8539,B 0.5627,C -0.0435,E1 0.4274,E2 306.4121} C_DIS
LIN {X -128.8965,Y 61.8952,Z 192,A 150.6595,B 0.563,C -0.0397,E1 0.4251,E2 304.5633} C_DIS
LIN {X -130.3665,Y 58.7363,Z 192,A 152.5672,B 0.5633,C -0.0357,E1 0.4228,E2 302.5975} C_DIS
LIN {X -132.1072,Y 54.7093,Z 192,A 154.7271,B 0.5635,C -0.0308,E1 0.4203,E2 300.3919} C_DIS
LIN {X -133.5003,Y 51.2183,Z 192,A 156.6612,B 0.5638,C -0.0264,E1 0.4183,E2 298.4084} C_DIS
LIN {X -134.6274,Y 48.1752,Z 192,A 158.3759,B 0.5639,C -0.0225,E1 0.4166,E2 296.6453} C_DIS
LIN {X -135.7659,Y 44.8665,Z 192,A 160.2155,B 0.5641,C -0.0182,E1 0.4149,E2 294.7541} C_DIS
LIN {X -136.8324,Y 41.5008,Z 192,A 162.0721,B 0.5642,C -0.0138,E1 0.4133,E2 292.8449} C_DIS
LIN {X -137.8284,Y 38.0636,Z 192,A 163.9648,B 0.5643,C -0.0093,E1 0.4118,E2 290.8971} C_DIS
LIN {X -138.7187,Y 34.6795,Z 192,A 165.8219,B 0.5643,C -0.0048,E1 0.4105,E2 288.9846} C_DIS
LIN {X -139.5243,Y 31.2826,Z 192,A 167.6805,B 0.5643,C -0.0003,E1 0.4093,E2 287.0697} C_DIS
LIN {X -140.2454,Y 27.8744,Z 192,A 169.6803,B 0.5643,C 0.0046,E1 0.4081,E2 284.9946} C_DIS
LIN {X -140.9457,Y 24.0824,Z 192,A 171.4723,B 0.5643,C 0.0092,E1 0.4072,E2 283.1722} C_DIS
LIN {X -141.4446,Y 20.9598,Z 192,A 173.3365,B 0.5643,C 0.0138,E1 0.4064,E2 281.2324} C_DIS
LIN {X -141.915,Y 17.4874,Z 192,A 175.2205,B 0.5641,C 0.0185,E1 0.4057,E2 279.2871} C_DIS
LIN {X -142.3001,Y 14.0054,Z 192,A 177.1282,B 0.5639,C 0.0234,E1 0.4051,E2 277.3144} C_DIS
LIN {X -142.5998,Y 10.5208,Z 192,A 178.9842,B 0.5637,C 0.0281,E1 0.4047,E2 275.3992} C_DIS
LIN {X -142.8157,Y 7.0066,Z 192,A -179.1249,B 0.5634,C 0.0329,E1 0.4044,E2 273.4453} C_DIS
LIN {X -142.9451,Y 3.5091,Z 192,A -177.2455,B 0.5631,C 0.0377,E1 0.4042,E2 271.5027} C_DIS
LIN {X -142.991,Y -0.0073,Z 192,A -175.2279,B 0.5628,C 0.0427,E1 0.4042,E2 269.4037} C_DIS
LIN {X -142.945,Y -3.5129,Z 192,A -173.4106,B 0.5624,C 0.0474,E1 0.4043,E2 267.5308} C_DIS
LIN {X -142.813,Y -7.0598,Z 192,A -171.5082,B 0.562,C 0.0522,E1 0.4045,E2 265.5631} C_DIS
LIN {X -142.5975,Y -10.5517,Z 192,A -169.6307,B 0.5615,C 0.057,E1 0.4049,E2 263.6203} C_DIS
LIN {X -142.2975,Y -14.0335,Z 192,A -167.754,B 0.561,C 0.0617,E1 0.4054,E2 261.6778} C_DIS
LIN {X -141.9123,Y -17.5099,Z 192,A -165.8777,B 0.5605,C 0.0663,E1 0.406,E2 259.7353} C_DIS
LIN {X -141.4427,Y -20.9735,Z 192,A -164.0013,B 0.5599,C 0.071,E1 0.4068,E2 257.7922} C_DIS
LIN {X -140.8869,Y -24.4297,Z 192,A -162.1026,B 0.5593,C 0.0756,E1 0.4077,E2 255.8233} C_DIS
LIN {X -140.2458,Y -27.8724,Z 192,A -160.0595,B 0.5586,C 0.0804,E1 0.4089,E2 253.6885} C_DIS
LIN {X -139.5146,Y -31.3251,Z 192,A -158.2906,B 0.558,C 0.0848,E1 0.41,E2 251.8688} C_DIS
LIN {X -138.7011,Y -34.7489,Z 192,A -156.5023,B 0.5573,C 0.089,E1 0.4112,E2 250.0259} C_DIS
LIN {X -137.8068,Y -38.141,Z 192,A -154.6538,B 0.5566,C 0.0934,E1 0.4126,E2 248.1129} C_DIS
LIN {X -136.8302,Y -41.508,Z 192,A -152.8126,B 0.5559,C 0.0976,E1 0.4141,E2 246.2079} C_DIS
LIN {X -135.7646,Y -44.8705,Z 192,A -150.9692,B 0.5551,C 0.1018,E1 0.4158,E2 244.3011} C_DIS
LIN {X -134.6248,Y -48.1824,Z 192,A -149.1209,B 0.5544,C 0.1059,E1 0.4176,E2 242.3868} C_DIS
LIN {X -133.4038,Y -51.4665,Z 192,A -147.3344,B 0.5536,C 0.1098,E1 0.4194,E2 240.5433} C_DIS
LIN {X -131.9922,Y -54.9847,Z 192,A -145.4598,B 0.5528,C 0.1139,E1 0.4215,E2 238.6156} C_DIS
LIN {X -130.7124,Y -57.963,Z 192,A -143.6856,B 0.552,C 0.1175,E1 0.4235,E2 236.7697} C_DIS
LIN {X -129.1344,Y -61.3971,Z 192,A -141.906,B 0.5512,C 0.1213,E1 0.4257,E2 234.9501} C_DIS
LIN {X -127.7217,Y -64.2869,Z 192,A -140.1694,B 0.5504,C 0.1247,E1 0.428,E2 233.1454} C_DIS
LIN {X -126.1004,Y -67.4136,Z 192,A -138.4009,B 0.5496,C 0.1281,E1 0.4304,E2 231.3223} C_DIS
LIN {X -124.4109,Y -70.4836,Z 192,A -136.6441,B 0.5489,C 0.1315,E1 0.4329,E2 229.5113} C_DIS
LIN {X -122.6461,Y -73.5111,Z 192,A -134.898,B 0.5481,C 0.1347,E1 0.4355,E2 227.7125} C_DIS
LIN {X -120.8077,Y -76.4942,Z 192,A -133.1719,B 0.5473,C 0.1378,E1 0.4382,E2 225.9365} C_DIS
LIN {X -118.8968,Y -79.4315,Z 192,A -131.4545,B 0.5465,C 0.1408,E1 0.441,E2 224.1704} C_DIS
LIN {X -116.9059,Y -82.3337,Z 192,A -129.6379,B 0.5458,C 0.1437,E1 0.444,E2 222.2902} C_DIS
LIN {X -114.3106,Y -85.901,Z 192,A -127.5207,B 0.5449,C 0.1472,E1 0.4477,E2 220.1182} C_DIS
LIN {X -111.6313,Y -89.3556,Z 192,A -125.5154,B 0.544,C 0.1503,E1 0.4513,E2 218.0731} C_DIS
LIN {X -109.4121,Y -92.0589,Z 192,A -123.8047,B 0.5433,C 0.1528,E1 0.4546,E2 216.3134} C_DIS
LIN {X -106.5305,Y -95.3785,Z 192,A -121.7957,B 0.5425,C 0.1557,E1 0.4585,E2 214.2652} C_DIS
LIN {X -104.1602,Y -97.9617,Z 192,A -120.0732,B 0.5418,C 0.1579,E1 0.4619,E2 212.492} C_DIS
LIN {X -101.0937,Y -101.124,Z 192,A -118.1124,B 0.5411,C 0.1605,E1 0.4659,E2 210.4999} C_DIS
LIN {X -98.5873,Y -103.5685,Z 192,A -116.5049,B 0.5405,C 0.1624,E1 0.4693,E2 208.8596} C_DIS
LIN {X -96.0228,Y -105.9502,Z 192,A -114.9141,B 0.54,C 0.1643,E1 0.4728,E2 207.2385} C_DIS
LIN {X -93.4008,Y -108.2687,Z 192,A -113.3349,B 0.5394,C 0.166,E1 0.4763,E2 205.6309} C_DIS
LIN {X -90.7236,Y -110.5221,Z 192,A -111.7617,B 0.5389,C 0.1676,E1 0.4798,E2 204.03} C_DIS
LIN {X -87.7675,Y -112.8837,Z 192,A -109.9547,B 0.5384,C 0.1691,E1 0.4841,E2 202.1757} C_DIS
LIN {X -84.4643,Y -115.3761,Z 192,A -108.2394,B 0.5379,C 0.1708,E1 0.4881,E2 200.451} C_DIS
LIN {X -81.6101,Y -117.4122,Z 192,A -106.7051,B 0.5375,C 0.172,E1 0.4918,E2 198.8955} C_DIS
LIN {X -78.5614,Y -119.4735,Z 192,A -104.974,B 0.5372,C 0.1731,E1 0.496,E2 197.1225} C_DIS
LIN {X -75.0134,Y -121.7329,Z 192,A -103.2918,B 0.5367,C 0.1744,E1 0.5002,E2 195.4406} C_DIS
LIN {X -72.0056,Y -123.5362,Z 192,A -101.7504,B 0.5365,C 0.1753,E1 0.5041,E2 193.8767} C_DIS
LIN {X -68.4085,Y -125.5631,Z 192,A -100.1548,B 0.5361,C 0.1764,E1 0.5081,E2 192.2903} C_DIS
LIN {X -65.8449,Y -126.9259,Z 192,A -98.7961,B 0.536,C 0.1769,E1 0.5117,E2 190.8995} C_DIS
LIN {X -62.7091,Y -128.5036,Z 192,A -97.3253,B 0.5357,C 0.1775,E1 0.5155,E2 189.4178} C_DIS
LIN {X -59.5356,Y -130.004,Z 192,A -95.8646,B 0.5356,C 0.178,E1 0.5194,E2 187.9478} C_DIS
LIN {X -56.3352,Y -131.4222,Z 192,A -94.4169,B 0.5354,C 0.1784,E1 0.5233,E2 186.4923} C_DIS
LIN {X -53.0982,Y -132.7629,Z 192,A -92.9679,B 0.5354,C 0.1788,E1 0.5272,E2 185.0354} C_DIS
LIN {X -49.0512,Y -134.3115,Z 192,A -91.3109,B 0.5352,C 0.1792,E1 0.5317,E2 183.3907} C_DIS
LIN {X -46.4798,Y -135.2222,Z 192,A -90.0883,B 0.5352,C 0.1792,E1 0.5351,E2 182.1466} C_DIS
LIN {X -43.1587,Y -136.3185,Z 192,A -88.6952,B 0.5352,C 0.1792,E1 0.539,E2 180.7543} C_DIS
LIN {X -39.8121,Y -137.3333,Z 192,A -87.2701,B 0.5352,C 0.1792,E1 0.543,E2 179.3246} C_DIS
LIN {X -36.4409,Y -138.2662,Z 192,A -85.891,B 0.5352,C 0.1792,E1 0.5469,E2 177.9486} C_DIS
LIN {X -33.0288,Y -139.121,Z 192,A -84.5126,B 0.5352,C 0.1791,E1 0.5507,E2 176.5746} C_DIS
LIN {X -29.4702,Y -139.919,Z 192,A -83.0852,B 0.5353,C 0.1788,E1 0.5548,E2 175.152} C_DIS
LIN {X -25.7733,Y -140.6464,Z 192,A -81.6951,B 0.5353,C 0.1786,E1 0.5587,E2 173.7808} C_DIS
LIN {X -22.7114,Y -141.1744,Z 192,A -80.3848,B 0.5356,C 0.1781,E1 0.5625,E2 172.4592} C_DIS
LIN {X -19.2467,Y -141.6876,Z 192,A -79.0232,B 0.5357,C 0.1776,E1 0.5664,E2 171.1037} C_DIS
LIN {X -15.747,Y -142.1182,Z 192,A -77.6758,B 0.5359,C 0.1771,E1 0.5703,E2 169.7661} C_DIS
LIN {X -12.2605,Y -142.4609,Z 192,A -76.3405,B 0.5361,C 0.1765,E1 0.5741,E2 168.4412} C_DIS
LIN {X -8.7631,Y -142.7186,Z 192,A -75.0137,B 0.5363,C 0.1758,E1 0.5779,E2 167.1264} C_DIS
LIN {X -5.264,Y -142.8908,Z 192,A -73.5664,B 0.5366,C 0.1748,E1 0.5821,E2 165.6711} C_DIS
LIN {X -1.7492,Y -142.9781,Z 192,A -72.3804,B 0.5368,C 0.1743,E1 0.5855,E2 164.5206} C_DIS
LIN {X 1.0259,Y -142.9828,Z 192,A -71.6241,B 0.5368,C 0.1743,E1 0.5875,E2 163.8216} C_DIS
Enddeposition()
LIN {X 1.0262,Y -143.032,Z 196.9998,A -71.6384,B 0.5368,C 0.1743,E1 0.5875,E2 163.8221} C_DIS
LIN {X 1.0272,Y -143.1798,Z 211.999,A -71.6848,B 0.537,C 0.1738,E1 0.5875,E2 163.8219} C_DIS
LIN {X 1.0272,Y -143.1798,Z 231.999,A -71.7616,B 0.5372,C 0.1731,E1 0.5875,E2 163.8213} C_DIS
END
